LIN {X -0.165,Y -561.534,Z 1075.002,A 0.000,B 0.000,C 90.000,E1 36.457} C_DIS
LIN {X 0.132,Y -558.565,Z 1074.998,A 0.000,B 0.000,C 90.000,E1 35.598} C_DIS
LIN {X 0.308,Y -556.320,Z 1074.995,A 0.000,B 0.000,C 90.000,E1 35.025} C_DIS
LIN {X 0.102,Y -552.086,Z 1074.989,A 0.000,B 0.000,C 90.000,E1 34.072} C_DIS
LIN {X 0.098,Y -548.792,Z 1074.985,A 0.000,B 0.000,C 90.000,E1 33.372} C_DIS
LIN {X 0.057,Y -545.238,Z 1074.982,A 0.000,B 0.000,C 90.000,E1 32.673} C_DIS
LIN {X 0.305,Y -540.806,Z 1074.977,A 0.000,B 0.000,C 90.000,E1 31.799} C_DIS
LIN {X -0.096,Y -536.840,Z 1074.973,A 0.000,B 0.000,C 90.000,E1 31.131} C_DIS
LIN {X -0.067,Y -532.563,Z 1074.969,A 0.000,B 0.000,C 90.000,E1 30.413} C_DIS
LIN {X 0.077,Y -528.884,Z 1074.966,A 0.000,B 0.000,C 90.000,E1 29.823} C_DIS
LIN {X -0.264,Y -524.894,Z 1074.963,A 0.000,B 0.000,C 90.000,E1 29.283} C_DIS
LIN {X 0.207,Y -518.481,Z 1074.958,A 0.000,B 0.000,C 90.000,E1 28.359} C_DIS
LIN {X 0.070,Y -512.632,Z 1074.954,A 0.000,B 0.000,C 90.000,E1 27.641} C_DIS
LIN {X -0.093,Y -506.270,Z 1074.950,A 0.000,B 0.000,C 90.000,E1 26.924} C_DIS
LIN {X -0.260,Y -500.914,Z 1074.946,A 0.000,B 0.000,C 90.000,E1 26.360} C_DIS
LIN {X 0.212,Y -494.053,Z 1074.942,A 0.000,B 0.000,C 90.000,E1 25.591} C_DIS
LIN {X 0.027,Y -485.704,Z 1074.938,A 0.000,B 0.000,C 90.000,E1 24.771} C_DIS
LIN {X 0.015,Y -475.699,Z 1074.932,A 0.000,B 0.000,C 90.000,E1 23.823} C_DIS
LIN {X 0.046,Y -466.824,Z 1074.928,A 0.000,B 0.000,C 90.000,E1 23.025} C_DIS
LIN {X -0.178,Y -453.420,Z 1074.922,A 0.000,B 0.000,C 90.000,E1 21.897} C_DIS
LIN {X -0.124,Y -431.292,Z 1074.910,A 0.000,B 0.000,C 90.000,E1 19.885} C_DIS
LIN {X -0.144,Y -418.613,Z 1074.903,A 0.000,B 0.000,C 90.000,E1 18.598} C_DIS
LIN {X -0.076,Y -409.051,Z 1074.897,A 0.000,B 0.000,C 90.000,E1 17.511} C_DIS
LIN {X 0.161,Y -401.164,Z 1074.892,A 0.000,B 0.000,C 90.000,E1 16.496} C_DIS
LIN {X 0.146,Y -397.859,Z 1074.889,A 0.000,B 0.000,C 90.000,E1 16.024} C_DIS
LIN {X 0.115,Y -396.044,Z 1074.888,A 0.000,B 0.000,C 90.000,E1 15.733} C_DIS
LIN {X -0.218,Y -395.141,Z 1074.887,A 0.000,B 0.000,C 90.000,E1 15.607} C_DIS
LIN {X -0.143,Y -393.859,Z 1074.885,A 0.000,B 0.000,C 90.000,E1 15.245} C_DIS
LIN {X -0.113,Y -393.096,Z 1074.884,A 0.000,B 0.000,C 90.000,E1 15.064} C_DIS
LIN {X -0.139,Y -392.054,Z 1074.881,A 0.000,B 0.000,C 90.000,E1 14.537} C_DIS
LIN {X -0.159,Y -391.808,Z 1074.877,A 0.000,B 0.000,C 90.000,E1 13.828} C_DIS
LIN {X -0.069,Y -392.415,Z 1074.873,A 0.000,B 0.000,C 90.000,E1 13.119} C_DIS
LIN {X 0.034,Y -399.707,Z 1074.847,A 0.000,B 0.000,C 90.000,E1 8.511} C_DIS
LIN {X -0.090,Y -404.135,Z 1074.836,A 0.000,B 0.000,C 90.000,E1 6.429} C_DIS
LIN {X -0.169,Y -407.950,Z 1074.826,A 0.000,B 0.000,C 90.000,E1 4.702} C_DIS
LIN {X -0.197,Y -408.866,Z 1074.824,A 0.000,B 0.000,C 90.000,E1 4.359} C_DIS
LIN {X -0.189,Y -410.221,Z 1074.822,A 0.000,B 0.000,C 90.000,E1 4.012} C_DIS
LIN {X -0.001,Y -412.147,Z 1074.820,A 0.000,B 0.000,C 90.000,E1 3.555} C_DIS
LIN {X -0.190,Y -416.804,Z 1074.816,A 0.000,B 0.000,C 90.000,E1 2.980} C_DIS
LIN {X 0.020,Y -417.622,Z 1074.816,A 0.000,B 0.000,C 90.000,E1 2.865} C_DIS
LIN {X 0.179,Y -422.679,Z 1074.814,A 0.000,B 0.000,C 90.000,E1 2.465} C_DIS
LIN {X -0.036,Y -434.410,Z 1074.810,A 0.000,B 0.000,C 90.000,E1 1.718} C_DIS
LIN {X 0.080,Y -459.258,Z 1074.801,A 0.000,B 0.000,C 90.000,E1 0.115} C_DIS
LIN {X -0.087,Y -474.381,Z 1074.796,A 0.000,B 0.000,C 90.000,E1 359.198} C_DIS
LIN {X 0.111,Y -484.224,Z 1074.792,A 0.000,B 0.000,C 90.000,E1 358.568} C_DIS
LIN {X -0.207,Y -495.380,Z 1074.788,A 0.000,B 0.000,C 90.000,E1 357.879} C_DIS
LIN {X 0.115,Y -503.194,Z 1074.785,A 0.000,B 0.000,C 90.000,E1 357.306} C_DIS
LIN {X 0.058,Y -510.520,Z 1074.782,A 0.000,B 0.000,C 90.000,E1 356.788} C_DIS
LIN {X 0.050,Y -516.476,Z 1074.780,A 0.000,B 0.000,C 90.000,E1 356.331} C_DIS
LIN {X -0.225,Y -523.750,Z 1074.776,A 0.000,B 0.000,C 90.000,E1 355.755} C_DIS
LIN {X 0.086,Y -531.946,Z 1074.772,A 0.000,B 0.000,C 90.000,E1 354.951} C_DIS
LIN {X -0.076,Y -537.186,Z 1074.769,A 0.000,B 0.000,C 90.000,E1 354.432} C_DIS
LIN {X -0.184,Y -543.345,Z 1074.765,A 0.000,B 0.000,C 90.000,E1 353.742} C_DIS
LIN {X -0.095,Y -548.003,Z 1074.762,A 0.000,B 0.000,C 90.000,E1 353.166} C_DIS
LIN {X -0.159,Y -553.081,Z 1074.758,A 0.000,B 0.000,C 90.000,E1 352.470} C_DIS
LIN {X 0.000,Y -556.784,Z 1074.755,A 0.000,B 0.000,C 90.000,E1 351.894} C_DIS
LIN {X -0.228,Y -561.640,Z 1074.750,A 0.000,B 0.000,C 90.000,E1 351.084} C_DIS
LIN {X 0.232,Y -563.986,Z 1074.748,A 0.000,B 0.000,C 90.000,E1 350.622} C_DIS
LIN {X -0.071,Y -568.640,Z 1074.743,A 0.000,B 0.000,C 90.000,E1 349.690} C_DIS
LIN {X -0.268,Y -571.076,Z 1074.740,A 0.000,B 0.000,C 90.000,E1 349.162} C_DIS
LIN {X 0.308,Y -574.633,Z 1074.735,A 0.000,B 0.000,C 90.000,E1 348.285} C_DIS
LIN {X 0.232,Y -580.028,Z 1074.728,A 0.000,B 0.000,C 90.000,E1 346.937} C_DIS
LIN {X 0.003,Y -584.013,Z 1074.722,A 0.000,B 0.000,C 90.000,E1 345.880} C_DIS
LIN {X -0.029,Y -587.800,Z 1074.716,A 0.000,B 0.000,C 90.000,E1 344.810} C_DIS
LIN {X 0.307,Y -590.501,Z 1074.711,A 0.000,B 0.000,C 90.000,E1 343.976} C_DIS
LIN {X 0.059,Y -594.876,Z 1074.704,A 0.000,B 0.000,C 90.000,E1 342.670} C_DIS
LIN {X -0.217,Y -598.220,Z 1074.698,A 0.000,B 0.000,C 90.000,E1 341.638} C_DIS
LIN {X -0.347,Y -600.546,Z 1074.693,A 0.000,B 0.000,C 90.000,E1 340.859} C_DIS
LIN {X -0.064,Y -604.004,Z 1074.686,A 0.000,B 0.000,C 90.000,E1 339.518} C_DIS
LIN {X 0.067,Y -605.993,Z 1074.682,A 0.000,B 0.000,C 90.000,E1 338.720} C_DIS
LIN {X 0.216,Y -607.758,Z 1074.677,A 0.000,B 0.000,C 90.000,E1 337.922} C_DIS
LIN {X 0.286,Y -610.437,Z 1074.670,A 0.000,B 0.000,C 90.000,E1 336.613} C_DIS
LIN {X -0.161,Y -612.623,Z 1074.663,A 0.000,B 0.000,C 90.000,E1 335.357} C_DIS
LIN {X 0.243,Y -614.458,Z 1074.656,A 0.000,B 0.000,C 90.000,E1 334.024} C_DIS
LIN {X 0.149,Y -615.747,Z 1074.650,A 0.000,B 0.000,C 90.000,E1 332.999} C_DIS
LIN {X 0.087,Y -616.628,Z 1074.646,A 0.000,B 0.000,C 90.000,E1 332.231} C_DIS
LIN {X 0.290,Y -617.753,Z 1074.639,A 0.000,B 0.000,C 90.000,E1 330.923} C_DIS
LIN {X -0.008,Y -618.335,Z 1074.633,A 0.000,B 0.000,C 90.000,E1 329.921} C_DIS
LIN {X 0.237,Y -618.642,Z 1074.627,A 0.000,B 0.000,C 90.000,E1 328.869} C_DIS
LIN {X -0.028,Y -618.644,Z 1074.623,A 0.000,B 0.000,C 90.000,E1 328.122} C_DIS
LIN {X -0.011,Y -618.295,Z 1074.616,A 0.000,B 0.000,C 90.000,E1 326.834} C_DIS
LIN {X 0.030,Y -617.634,Z 1074.610,A 0.000,B 0.000,C 90.000,E1 325.801} C_DIS
LIN {X 0.102,Y -617.036,Z 1074.606,A 0.000,B 0.000,C 90.000,E1 325.022} C_DIS
LIN {X -0.013,Y -615.176,Z 1074.594,A 0.000,B 0.000,C 90.000,E1 322.970} C_DIS
LIN {X 0.069,Y -614.027,Z 1074.586,A 0.000,B 0.000,C 90.000,E1 321.412} C_DIS
LIN {X -0.062,Y -612.361,Z 1074.573,A 0.000,B 0.000,C 90.000,E1 319.094} C_DIS
LIN {X -0.035,Y -611.598,Z 1074.566,A 0.000,B 0.000,C 90.000,E1 317.796} C_DIS
LIN {X -0.388,Y -611.230,Z 1074.563,A 0.000,B 0.000,C 90.000,E1 317.310} C_DIS
LIN {X -0.323,Y -609.621,Z 1074.553,A 0.000,B 0.000,C 90.000,E1 315.486} C_DIS
LIN {X -0.060,Y -607.968,Z 1074.541,A 0.000,B 0.000,C 90.000,E1 313.380} C_DIS
LIN {X -0.301,Y -606.609,Z 1074.532,A 0.000,B 0.000,C 90.000,E1 311.838} C_DIS
LIN {X -0.108,Y -605.128,Z 1074.524,A 0.000,B 0.000,C 90.000,E1 310.253} C_DIS
LIN {X 0.001,Y -604.301,Z 1074.518,A 0.000,B 0.000,C 90.000,E1 309.197} C_DIS
LIN {X 0.049,Y -603.773,Z 1074.515,A 0.000,B 0.000,C 90.000,E1 308.669} C_DIS
LIN {X -0.025,Y -603.222,Z 1074.510,A 0.000,B 0.000,C 90.000,E1 307.890} C_DIS
LIN {X -0.408,Y -601.658,Z 1074.500,A 0.000,B 0.000,C 90.000,E1 306.091} C_DIS
LIN {X 0.341,Y -600.780,Z 1074.496,A 0.000,B 0.000,C 90.000,E1 305.231} C_DIS
LIN {X -0.102,Y -599.901,Z 1074.492,A 0.000,B 0.000,C 90.000,E1 304.485} C_DIS
LIN {X 0.158,Y -597.860,Z 1074.483,A 0.000,B 0.000,C 90.000,E1 302.880} C_DIS
LIN {X 0.197,Y -596.605,Z 1074.478,A 0.000,B 0.000,C 90.000,E1 302.084} C_DIS
LIN {X -0.183,Y -595.601,Z 1074.475,A 0.000,B 0.000,C 90.000,E1 301.592} C_DIS
LIN {X -0.163,Y -593.715,Z 1074.471,A 0.000,B 0.000,C 90.000,E1 300.797} C_DIS
LIN {X -0.160,Y -591.348,Z 1074.467,A 0.000,B 0.000,C 90.000,E1 300.001} C_DIS
LIN {X -0.182,Y -588.499,Z 1074.462,A 0.000,B 0.000,C 90.000,E1 299.205} C_DIS
LIN {X 0.217,Y -584.185,Z 1074.457,A 0.000,B 0.000,C 90.000,E1 298.231} C_DIS
LIN {X 0.032,Y -581.939,Z 1074.455,A 0.000,B 0.000,C 90.000,E1 297.847} C_DIS
LIN {X -0.163,Y -579.429,Z 1074.453,A 0.000,B 0.000,C 90.000,E1 297.462} C_DIS
LIN {X -0.178,Y -575.517,Z 1074.450,A 0.000,B 0.000,C 90.000,E1 296.924} C_DIS
LIN {X 0.185,Y -573.298,Z 1074.448,A 0.000,B 0.000,C 90.000,E1 296.616} C_DIS
LIN {X 0.109,Y -571.984,Z 1074.447,A 0.000,B 0.000,C 90.000,E1 296.488} C_DIS
LIN {X 0.021,Y -568.906,Z 1074.446,A 0.000,B 0.000,C 90.000,E1 296.232} C_DIS
LIN {X 0.165,Y -565.892,Z 1074.444,A 0.000,B 0.000,C 90.000,E1 295.976} C_DIS
LIN {X 0.274,Y -564.016,Z 1074.444,A 0.000,B 0.000,C 90.000,E1 295.848} C_DIS
LIN {X -0.123,Y -561.660,Z 1074.443,A 0.000,B 0.000,C 90.000,E1 295.771} C_DIS
LIN {X 0.029,Y -557.315,Z 1074.442,A 0.000,B 0.000,C 90.000,E1 295.591} C_DIS
LIN {X 0.071,Y -554.762,Z 1074.442,A 0.000,B 0.000,C 90.000,E1 295.463} C_DIS
LIN {X -0.158,Y -552.795,Z 1074.441,A 0.000,B 0.000,C 90.000,E1 295.412} C_DIS
LIN {X -0.148,Y -551.370,Z 1074.441,A 0.000,B 0.000,C 90.000,E1 295.335} C_DIS
LIN {X 0.171,Y -549.416,Z 1074.440,A 0.000,B 0.000,C 90.000,E1 295.155} C_DIS
LIN {X -0.319,Y -547.636,Z 1074.439,A 0.000,B 0.000,C 90.000,E1 295.027} C_DIS
LIN {X 0.122,Y -546.552,Z 1074.438,A 0.000,B 0.000,C 90.000,E1 294.847} C_DIS
LIN {X -0.055,Y -545.055,Z 1074.437,A 0.000,B 0.000,C 90.000,E1 294.591} C_DIS
LIN {X 0.068,Y -543.671,Z 1074.434,A 0.000,B 0.000,C 90.000,E1 294.155} C_DIS
LIN {X -0.264,Y -543.036,Z 1074.432,A 0.000,B 0.000,C 90.000,E1 293.770} C_DIS
LIN {X -0.282,Y -542.679,Z 1074.429,A 0.000,B 0.000,C 90.000,E1 293.206} C_DIS
LIN {X 0.170,Y -542.511,Z 1074.422,A 0.000,B 0.000,C 90.000,E1 292.025} C_DIS
LIN {X -0.088,Y -542.359,Z 1074.416,A 0.000,B 0.000,C 90.000,E1 290.918} C_DIS
LIN {X -0.060,Y -542.525,Z 1074.407,A 0.000,B 0.000,C 90.000,E1 289.214} C_DIS
LIN {X 0.186,Y -542.645,Z 1074.401,A 0.000,B 0.000,C 90.000,E1 288.055} C_DIS
LIN {X 0.259,Y -542.719,Z 1074.394,A 0.000,B 0.000,C 90.000,E1 286.913} C_DIS
LIN {X -0.121,Y -542.449,Z 1074.386,A 0.000,B 0.000,C 90.000,E1 285.536} C_DIS
LIN {X -0.128,Y -541.988,Z 1074.378,A 0.000,B 0.000,C 90.000,E1 284.120} C_DIS
LIN {X -0.143,Y -541.426,Z 1074.370,A 0.000,B 0.000,C 90.000,E1 282.703} C_DIS
LIN {X -0.215,Y -540.575,Z 1074.361,A 0.000,B 0.000,C 90.000,E1 281.007} C_DIS
LIN {X 0.198,Y -539.496,Z 1074.350,A 0.000,B 0.000,C 90.000,E1 278.973} C_DIS
LIN {X -0.094,Y -538.562,Z 1074.341,A 0.000,B 0.000,C 90.000,E1 277.296} C_DIS
LIN {X 0.069,Y -537.801,Z 1074.333,A 0.000,B 0.000,C 90.000,E1 275.853} C_DIS
LIN {X 0.207,Y -536.736,Z 1074.322,A 0.000,B 0.000,C 90.000,E1 273.841} C_DIS
LIN {X 0.259,Y -535.709,Z 1074.310,A 0.000,B 0.000,C 90.000,E1 271.835} C_DIS
LIN {X -0.247,Y -534.783,Z 1074.301,A 0.000,B 0.000,C 90.000,E1 270.172} C_DIS
LIN {X -0.249,Y -533.966,Z 1074.293,A 0.000,B 0.000,C 90.000,E1 268.740} C_DIS
LIN {X -0.248,Y -533.309,Z 1074.286,A 0.000,B 0.000,C 90.000,E1 267.593} C_DIS
LIN {X -0.242,Y -532.307,Z 1074.277,A 0.000,B 0.000,C 90.000,E1 265.869} C_DIS
LIN {X -0.240,Y -531.249,Z 1074.269,A 0.000,B 0.000,C 90.000,E1 264.432} C_DIS
LIN {X -0.205,Y -529.945,Z 1074.261,A 0.000,B 0.000,C 90.000,E1 262.989} C_DIS
LIN {X -0.196,Y -528.468,Z 1074.253,A 0.000,B 0.000,C 90.000,E1 261.546} C_DIS
LIN {X -0.093,Y -526.288,Z 1074.242,A 0.000,B 0.000,C 90.000,E1 259.511} C_DIS
LIN {X 0.050,Y -524.135,Z 1074.230,A 0.000,B 0.000,C 90.000,E1 257.465} C_DIS
LIN {X 0.230,Y -522.650,Z 1074.222,A 0.000,B 0.000,C 90.000,E1 255.992} C_DIS
LIN {X 0.008,Y -520.608,Z 1074.211,A 0.000,B 0.000,C 90.000,E1 253.976} C_DIS
LIN {X -0.111,Y -518.750,Z 1074.201,A 0.000,B 0.000,C 90.000,E1 252.236} C_DIS
LIN {X 0.111,Y -517.533,Z 1074.195,A 0.000,B 0.000,C 90.000,E1 251.040} C_DIS
LIN {X 0.122,Y -515.892,Z 1074.187,A 0.000,B 0.000,C 90.000,E1 249.571} C_DIS
LIN {X 0.104,Y -514.022,Z 1074.178,A 0.000,B 0.000,C 90.000,E1 248.103} C_DIS
LIN {X -0.116,Y -511.574,Z 1074.169,A 0.000,B 0.000,C 90.000,E1 246.357} C_DIS
LIN {X 0.181,Y -509.315,Z 1074.160,A 0.000,B 0.000,C 90.000,E1 244.845} C_DIS
LIN {X -0.026,Y -506.957,Z 1074.152,A 0.000,B 0.000,C 90.000,E1 243.384} C_DIS
LIN {X 0.320,Y -504.954,Z 1074.146,A 0.000,B 0.000,C 90.000,E1 242.153} C_DIS
LIN {X 0.121,Y -501.896,Z 1074.136,A 0.000,B 0.000,C 90.000,E1 240.383} C_DIS
LIN {X -0.154,Y -498.729,Z 1074.126,A 0.000,B 0.000,C 90.000,E1 238.614} C_DIS
LIN {X 0.006,Y -495.417,Z 1074.115,A 0.000,B 0.000,C 90.000,E1 236.786} C_DIS
LIN {X -0.048,Y -491.856,Z 1074.105,A 0.000,B 0.000,C 90.000,E1 234.975} C_DIS
LIN {X 0.265,Y -488.776,Z 1074.097,A 0.000,B 0.000,C 90.000,E1 233.417} C_DIS
LIN {X 0.127,Y -485.562,Z 1074.089,A 0.000,B 0.000,C 90.000,E1 231.904} C_DIS
LIN {X 0.043,Y -481.501,Z 1074.078,A 0.000,B 0.000,C 90.000,E1 230.070} C_DIS
LIN {X -0.183,Y -475.565,Z 1074.063,A 0.000,B 0.000,C 90.000,E1 227.310} C_DIS
LIN {X -0.052,Y -470.828,Z 1074.049,A 0.000,B 0.000,C 90.000,E1 224.798} C_DIS
LIN {X 0.034,Y -467.996,Z 1074.040,A 0.000,B 0.000,C 90.000,E1 223.218} C_DIS
LIN {X -0.248,Y -464.960,Z 1074.031,A 0.000,B 0.000,C 90.000,E1 221.676} C_DIS
LIN {X 0.161,Y -461.136,Z 1074.021,A 0.000,B 0.000,C 90.000,E1 219.725} C_DIS
LIN {X -0.192,Y -458.057,Z 1074.012,A 0.000,B 0.000,C 90.000,E1 218.177} C_DIS
LIN {X -0.244,Y -454.887,Z 1074.003,A 0.000,B 0.000,C 90.000,E1 216.583} C_DIS
LIN {X -0.204,Y -450.241,Z 1073.991,A 0.000,B 0.000,C 90.000,E1 214.326} C_DIS
LIN {X 0.198,Y -445.779,Z 1073.978,A 0.000,B 0.000,C 90.000,E1 212.005} C_DIS
LIN {X 0.071,Y -443.385,Z 1073.971,A 0.000,B 0.000,C 90.000,E1 210.718} C_DIS
LIN {X 0.111,Y -440.255,Z 1073.962,A 0.000,B 0.000,C 90.000,E1 209.077} C_DIS
LIN {X -0.087,Y -436.535,Z 1073.951,A 0.000,B 0.000,C 90.000,E1 207.129} C_DIS
LIN {X -0.175,Y -433.150,Z 1073.940,A 0.000,B 0.000,C 90.000,E1 205.155} C_DIS
LIN {X -0.144,Y -429.512,Z 1073.927,A 0.000,B 0.000,C 90.000,E1 202.823} C_DIS
LIN {X 0.044,Y -426.761,Z 1073.916,A 0.000,B 0.000,C 90.000,E1 200.791} C_DIS
LIN {X -0.162,Y -425.837,Z 1073.910,A 0.000,B 0.000,C 90.000,E1 199.812} C_DIS
LIN {X -0.173,Y -425.484,Z 1073.906,A 0.000,B 0.000,C 90.000,E1 199.141} C_DIS
LIN {X 0.215,Y -425.212,Z 1073.902,A 0.000,B 0.000,C 90.000,E1 198.417} C_DIS
LIN {X 0.065,Y -425.334,Z 1073.899,A 0.000,B 0.000,C 90.000,E1 197.764} C_DIS
LIN {X 0.046,Y -425.808,Z 1073.895,A 0.000,B 0.000,C 90.000,E1 197.094} C_DIS
LIN {X -0.097,Y -426.809,Z 1073.891,A 0.000,B 0.000,C 90.000,E1 196.441} C_DIS
LIN {X -0.031,Y -429.236,Z 1073.886,A 0.000,B 0.000,C 90.000,E1 195.426} C_DIS
LIN {X -0.044,Y -431.990,Z 1073.881,A 0.000,B 0.000,C 90.000,E1 194.592} C_DIS
LIN {X 0.006,Y -439.992,Z 1073.871,A 0.000,B 0.000,C 90.000,E1 192.771} C_DIS
LIN {X -0.216,Y -450.151,Z 1073.860,A 0.000,B 0.000,C 90.000,E1 190.838} C_DIS
LIN {X 0.164,Y -461.062,Z 1073.849,A 0.000,B 0.000,C 90.000,E1 188.859} C_DIS
LIN {X 0.192,Y -468.397,Z 1073.842,A 0.000,B 0.000,C 90.000,E1 187.587} C_DIS
LIN {X 0.039,Y -473.849,Z 1073.837,A 0.000,B 0.000,C 90.000,E1 186.663} C_DIS
LIN {X -0.057,Y -479.015,Z 1073.832,A 0.000,B 0.000,C 90.000,E1 185.739} C_DIS
LIN {X 0.044,Y -484.844,Z 1073.826,A 0.000,B 0.000,C 90.000,E1 184.645} C_DIS
LIN {X 0.026,Y -489.888,Z 1073.821,A 0.000,B 0.000,C 90.000,E1 183.726} C_DIS
LIN {X 0.238,Y -495.579,Z 1073.815,A 0.000,B 0.000,C 90.000,E1 182.636} C_DIS
LIN {X 0.028,Y -501.228,Z 1073.809,A 0.000,B 0.000,C 90.000,E1 181.604} C_DIS
LIN {X 0.075,Y -507.486,Z 1073.802,A 0.000,B 0.000,C 90.000,E1 180.401} C_DIS
LIN {X 0.142,Y -515.276,Z 1073.794,A 0.000,B 0.000,C 90.000,E1 178.912} C_DIS
LIN {X 0.184,Y -520.701,Z 1073.788,A 0.000,B 0.000,C 90.000,E1 177.879} C_DIS
LIN {X -0.044,Y -529.758,Z 1073.779,A 0.000,B 0.000,C 90.000,E1 176.159} C_DIS
LIN {X -0.007,Y -538.730,Z 1073.769,A 0.000,B 0.000,C 90.000,E1 174.432} C_DIS
LIN {X -0.051,Y -546.842,Z 1073.760,A 0.000,B 0.000,C 90.000,E1 172.875} C_DIS
LIN {X 0.198,Y -552.617,Z 1073.754,A 0.000,B 0.000,C 90.000,E1 171.724} C_DIS
LIN {X 0.055,Y -558.314,Z 1073.748,A 0.000,B 0.000,C 90.000,E1 170.622} C_DIS
LIN {X -0.160,Y -564.503,Z 1073.741,A 0.000,B 0.000,C 90.000,E1 169.398} C_DIS
LIN {X 0.102,Y -569.230,Z 1073.736,A 0.000,B 0.000,C 90.000,E1 168.409} C_DIS
LIN {X 0.100,Y -573.086,Z 1073.731,A 0.000,B 0.000,C 90.000,E1 167.589} C_DIS
LIN {X -0.211,Y -580.574,Z 1073.722,A 0.000,B 0.000,C 90.000,E1 165.992} C_DIS
LIN {X -0.191,Y -584.733,Z 1073.717,A 0.000,B 0.000,C 90.000,E1 165.046} C_DIS
LIN {X 0.111,Y -588.117,Z 1073.712,A 0.000,B 0.000,C 90.000,E1 164.212} C_DIS
LIN {X 0.141,Y -592.450,Z 1073.706,A 0.000,B 0.000,C 90.000,E1 163.142} C_DIS
LIN {X -0.042,Y -595.527,Z 1073.702,A 0.000,B 0.000,C 90.000,E1 162.362} C_DIS
LIN {X 0.264,Y -599.459,Z 1073.696,A 0.000,B 0.000,C 90.000,E1 161.275} C_DIS
LIN {X -0.232,Y -604.018,Z 1073.689,A 0.000,B 0.000,C 90.000,E1 160.007} C_DIS
LIN {X -0.103,Y -606.577,Z 1073.684,A 0.000,B 0.000,C 90.000,E1 159.209} C_DIS
LIN {X -0.280,Y -610.636,Z 1073.677,A 0.000,B 0.000,C 90.000,E1 157.922} C_DIS
LIN {X 0.151,Y -613.007,Z 1073.673,A 0.000,B 0.000,C 90.000,E1 157.102} C_DIS
LIN {X 0.319,Y -616.607,Z 1073.666,A 0.000,B 0.000,C 90.000,E1 155.793} C_DIS
LIN {X -0.030,Y -620.754,Z 1073.657,A 0.000,B 0.000,C 90.000,E1 154.280} C_DIS
LIN {X -0.031,Y -624.543,Z 1073.649,A 0.000,B 0.000,C 90.000,E1 152.743} C_DIS
LIN {X 0.007,Y -627.078,Z 1073.643,A 0.000,B 0.000,C 90.000,E1 151.719} C_DIS
LIN {X -0.174,Y -629.490,Z 1073.637,A 0.000,B 0.000,C 90.000,E1 150.717} C_DIS
LIN {X -0.259,Y -632.942,Z 1073.629,A 0.000,B 0.000,C 90.000,E1 149.203} C_DIS
LIN {X 0.074,Y -636.745,Z 1073.619,A 0.000,B 0.000,C 90.000,E1 147.406} C_DIS
LIN {X -0.238,Y -640.357,Z 1073.609,A 0.000,B 0.000,C 90.000,E1 145.674} C_DIS
LIN {X 0.018,Y -643.392,Z 1073.601,A 0.000,B 0.000,C 90.000,E1 144.149} C_DIS
LIN {X 0.189,Y -646.342,Z 1073.593,A 0.000,B 0.000,C 90.000,E1 142.637} C_DIS
LIN {X 0.045,Y -647.872,Z 1073.588,A 0.000,B 0.000,C 90.000,E1 141.904} C_DIS
LIN {X 0.281,Y -650.336,Z 1073.582,A 0.000,B 0.000,C 90.000,E1 140.642} C_DIS
LIN {X 0.030,Y -653.843,Z 1073.572,A 0.000,B 0.000,C 90.000,E1 138.933} C_DIS
LIN {X -0.173,Y -656.959,Z 1073.564,A 0.000,B 0.000,C 90.000,E1 137.472} C_DIS
LIN {X 0.089,Y -661.271,Z 1073.553,A 0.000,B 0.000,C 90.000,E1 135.486} C_DIS
LIN {X 0.009,Y -664.876,Z 1073.545,A 0.000,B 0.000,C 90.000,E1 134.028} C_DIS
LIN {X 0.028,Y -669.235,Z 1073.535,A 0.000,B 0.000,C 90.000,E1 132.324} C_DIS
LIN {X 0.138,Y -673.000,Z 1073.527,A 0.000,B 0.000,C 90.000,E1 130.862} C_DIS
LIN {X -0.123,Y -676.778,Z 1073.519,A 0.000,B 0.000,C 90.000,E1 129.439} C_DIS
LIN {X -0.158,Y -681.668,Z 1073.508,A 0.000,B 0.000,C 90.000,E1 127.523} C_DIS
LIN {X -0.342,Y -684.154,Z 1073.503,A 0.000,B 0.000,C 90.000,E1 126.583} C_DIS
LIN {X -0.124,Y -686.021,Z 1073.499,A 0.000,B 0.000,C 90.000,E1 125.851} C_DIS
LIN {X -0.079,Y -688.857,Z 1073.493,A 0.000,B 0.000,C 90.000,E1 124.659} C_DIS
LIN {X 0.203,Y -691.761,Z 1073.486,A 0.000,B 0.000,C 90.000,E1 123.452} C_DIS
LIN {X -0.266,Y -694.068,Z 1073.481,A 0.000,B 0.000,C 90.000,E1 122.546} C_DIS
LIN {X 0.223,Y -695.750,Z 1073.477,A 0.000,B 0.000,C 90.000,E1 121.799} C_DIS
LIN {X -0.324,Y -698.389,Z 1073.470,A 0.000,B 0.000,C 90.000,E1 120.669} C_DIS
LIN {X 0.201,Y -699.820,Z 1073.466,A 0.000,B 0.000,C 90.000,E1 119.922} C_DIS
LIN {X 0.391,Y -700.876,Z 1073.463,A 0.000,B 0.000,C 90.000,E1 119.205} C_DIS
LIN {X 0.318,Y -701.494,Z 1073.460,A 0.000,B 0.000,C 90.000,E1 118.743} C_DIS
LIN {X 0.002,Y -703.478,Z 1073.448,A 0.000,B 0.000,C 90.000,E1 116.668} C_DIS
LIN {X 0.194,Y -704.395,Z 1073.443,A 0.000,B 0.000,C 90.000,E1 115.720} C_DIS
LIN {X -0.173,Y -704.786,Z 1073.440,A 0.000,B 0.000,C 90.000,E1 115.283} C_DIS
LIN {X -0.238,Y -704.963,Z 1073.438,A 0.000,B 0.000,C 90.000,E1 114.823} C_DIS
LIN {X -0.245,Y -704.961,Z 1073.437,A 0.000,B 0.000,C 90.000,E1 114.591} C_DIS
LIN {X 0.328,Y -704.505,Z 1073.434,A 0.000,B 0.000,C 90.000,E1 114.079} C_DIS
LIN {X -0.316,Y -703.985,Z 1073.433,A 0.000,B 0.000,C 90.000,E1 113.898} C_DIS
LIN {X 0.248,Y -702.448,Z 1073.430,A 0.000,B 0.000,C 90.000,E1 113.387} C_DIS
LIN {X 0.386,Y -701.844,Z 1073.429,A 0.000,B 0.000,C 90.000,E1 113.259} C_DIS
LIN {X 0.007,Y -698.300,Z 1073.427,A 0.000,B 0.000,C 90.000,E1 112.823} C_DIS
LIN {X -0.131,Y -697.259,Z 1073.426,A 0.000,B 0.000,C 90.000,E1 112.717} C_DIS
LIN {X -0.001,Y -695.687,Z 1073.426,A 0.000,B 0.000,C 90.000,E1 112.589} C_DIS
LIN {X -0.164,Y -688.279,Z 1073.424,A 0.000,B 0.000,C 90.000,E1 112.259} C_DIS
LIN {X 0.227,Y -686.446,Z 1073.423,A 0.000,B 0.000,C 90.000,E1 112.153} C_DIS
LIN {X 0.128,Y -684.148,Z 1073.423,A 0.000,B 0.000,C 90.000,E1 112.099} C_DIS
LIN {X -0.175,Y -676.156,Z 1073.422,A 0.000,B 0.000,C 90.000,E1 112.025} C_DIS
LIN {X -0.205,Y -607.048,Z 1073.422,A 0.000,B 0.000,C 90.000,E1 112.025} C_DIS
LIN {X 0.255,Y -601.997,Z 1073.421,A 0.000,B 0.000,C 90.000,E1 111.770} C_DIS
LIN {X 0.315,Y -596.175,Z 1073.419,A 0.000,B 0.000,C 90.000,E1 111.408} C_DIS
LIN {X 0.074,Y -588.927,Z 1073.416,A 0.000,B 0.000,C 90.000,E1 110.865} C_DIS
LIN {X 0.166,Y -580.721,Z 1073.412,A 0.000,B 0.000,C 90.000,E1 110.174} C_DIS
LIN {X 0.161,Y -575.155,Z 1073.410,A 0.000,B 0.000,C 90.000,E1 109.704} C_DIS
LIN {X 0.085,Y -569.130,Z 1073.407,A 0.000,B 0.000,C 90.000,E1 109.268} C_DIS
LIN {X -0.122,Y -560.870,Z 1073.404,A 0.000,B 0.000,C 90.000,E1 108.779} C_DIS
LIN {X -0.172,Y -554.271,Z 1073.402,A 0.000,B 0.000,C 90.000,E1 108.417} C_DIS
LIN {X 0.050,Y -549.376,Z 1073.400,A 0.000,B 0.000,C 90.000,E1 108.055} C_DIS
LIN {X -0.163,Y -547.701,Z 1073.399,A 0.000,B 0.000,C 90.000,E1 107.873} C_DIS
LIN {X -0.205,Y -547.669,Z 1073.399,A 0.000,B 0.000,C 90.000,E1 107.873} C_DIS
LIN {X -0.176,Y -547.352,Z 1073.398,A 0.000,B 0.000,C 90.000,E1 107.638} C_DIS
LIN {X 0.157,Y -547.444,Z 1073.395,A 0.000,B 0.000,C 90.000,E1 107.040} C_DIS
LIN {X -0.130,Y -548.416,Z 1073.387,A 0.000,B 0.000,C 90.000,E1 105.662} C_DIS
LIN {X -0.105,Y -549.993,Z 1073.375,A 0.000,B 0.000,C 90.000,E1 103.411} C_DIS
LIN {X 0.256,Y -551.925,Z 1073.362,A 0.000,B 0.000,C 90.000,E1 101.130} C_DIS
LIN {X 0.034,Y -554.290,Z 1073.350,A 0.000,B 0.000,C 90.000,E1 98.916} C_DIS
LIN {X 0.073,Y -556.176,Z 1073.340,A 0.000,B 0.000,C 90.000,E1 97.239} C_DIS
LIN {X 0.020,Y -557.718,Z 1073.333,A 0.000,B 0.000,C 90.000,E1 95.853} C_DIS
LIN {X -0.066,Y -559.077,Z 1073.325,A 0.000,B 0.000,C 90.000,E1 94.473} C_DIS
LIN {X -0.132,Y -559.941,Z 1073.317,A 0.000,B 0.000,C 90.000,E1 93.094} C_DIS
LIN {X -0.220,Y -560.677,Z 1073.309,A 0.000,B 0.000,C 90.000,E1 91.718} C_DIS
LIN {X -0.208,Y -561.466,Z 1073.300,A 0.000,B 0.000,C 90.000,E1 90.057} C_DIS
LIN {X -0.180,Y -562.039,Z 1073.291,A 0.000,B 0.000,C 90.000,E1 88.396} C_DIS
LIN {X -0.101,Y -562.696,Z 1073.282,A 0.000,B 0.000,C 90.000,E1 86.731} C_DIS
LIN {X -0.139,Y -563.235,Z 1073.274,A 0.000,B 0.000,C 90.000,E1 85.355} C_DIS
LIN {X 0.015,Y -563.758,Z 1073.265,A 0.000,B 0.000,C 90.000,E1 83.685} C_DIS
LIN {X 0.252,Y -564.259,Z 1073.256,A 0.000,B 0.000,C 90.000,E1 82.008} C_DIS
LIN {X 0.171,Y -564.524,Z 1073.250,A 0.000,B 0.000,C 90.000,E1 80.914} C_DIS
LIN {X -0.116,Y -565.090,Z 1073.242,A 0.000,B 0.000,C 90.000,E1 79.567} C_DIS
LIN {X 0.233,Y -565.824,Z 1073.233,A 0.000,B 0.000,C 90.000,E1 77.881} C_DIS
LIN {X -0.098,Y -566.875,Z 1073.222,A 0.000,B 0.000,C 90.000,E1 75.992} C_DIS
LIN {X 0.044,Y -568.982,Z 1073.205,A 0.000,B 0.000,C 90.000,E1 72.960} C_DIS
LIN {X 0.099,Y -570.513,Z 1073.195,A 0.000,B 0.000,C 90.000,E1 71.040} C_DIS
LIN {X 0.032,Y -572.135,Z 1073.184,A 0.000,B 0.000,C 90.000,E1 69.135} C_DIS
LIN {X 0.010,Y -573.674,Z 1073.174,A 0.000,B 0.000,C 90.000,E1 67.230} C_DIS
LIN {X -0.136,Y -574.960,Z 1073.165,A 0.000,B 0.000,C 90.000,E1 65.613} C_DIS
LIN {X -0.026,Y -575.984,Z 1073.155,A 0.000,B 0.000,C 90.000,E1 63.973} C_DIS
LIN {X -0.159,Y -576.937,Z 1073.146,A 0.000,B 0.000,C 90.000,E1 62.359} C_DIS
LIN {X 0.006,Y -577.832,Z 1073.137,A 0.000,B 0.000,C 90.000,E1 60.717} C_DIS
LIN {X 0.341,Y -578.490,Z 1073.130,A 0.000,B 0.000,C 90.000,E1 59.331} C_DIS
LIN {X 0.186,Y -579.098,Z 1073.122,A 0.000,B 0.000,C 90.000,E1 57.995} C_DIS
LIN {X 0.190,Y -579.849,Z 1073.113,A 0.000,B 0.000,C 90.000,E1 56.373} C_DIS
LIN {X 0.044,Y -580.513,Z 1073.104,A 0.000,B 0.000,C 90.000,E1 54.769} C_DIS
LIN {X -0.090,Y -580.799,Z 1073.098,A 0.000,B 0.000,C 90.000,E1 53.703} C_DIS
LIN {X -0.050,Y -581.040,Z 1073.091,A 0.000,B 0.000,C 90.000,E1 52.351} C_DIS
LIN {X 0.006,Y -580.977,Z 1073.086,A 0.000,B 0.000,C 90.000,E1 51.537} C_DIS
LIN {X 0.064,Y -580.869,Z 1073.082,A 0.000,B 0.000,C 90.000,E1 50.723} C_DIS
LIN {X 0.009,Y -580.452,Z 1073.074,A 0.000,B 0.000,C 90.000,E1 49.380} C_DIS
LIN {X -0.219,Y -580.027,Z 1073.068,A 0.000,B 0.000,C 90.000,E1 48.324} C_DIS
LIN {X -0.067,Y -579.457,Z 1073.062,A 0.000,B 0.000,C 90.000,E1 47.229} C_DIS
LIN {X -0.198,Y -578.610,Z 1073.055,A 0.000,B 0.000,C 90.000,E1 45.891} C_DIS
LIN {X -0.074,Y -577.673,Z 1073.049,A 0.000,B 0.000,C 90.000,E1 44.798} C_DIS
LIN {X 0.318,Y -576.792,Z 1073.044,A 0.000,B 0.000,C 90.000,E1 43.947} C_DIS
LIN {X 0.000,Y -575.375,Z 1073.038,A 0.000,B 0.000,C 90.000,E1 42.894} C_DIS
LIN {X 0.211,Y -573.401,Z 1073.031,A 0.000,B 0.000,C 90.000,E1 41.515} C_DIS
LIN {X -0.117,Y -571.371,Z 1073.025,A 0.000,B 0.000,C 90.000,E1 40.458} C_DIS
LIN {X 0.147,Y -570.322,Z 1073.022,A 0.000,B 0.000,C 90.000,E1 39.886} C_DIS
LIN {X -0.221,Y -567.791,Z 1073.016,A 0.000,B 0.000,C 90.000,E1 38.830} C_DIS
LIN {X 0.144,Y -565.719,Z 1073.011,A 0.000,B 0.000,C 90.000,E1 37.971} C_DIS
LIN {X 0.039,Y -563.336,Z 1073.006,A 0.000,B 0.000,C 90.000,E1 37.156} C_DIS
LIN {X 0.252,Y -561.570,Z 1073.003,A 0.000,B 0.000,C 90.000,E1 36.583} C_DIS
LIN {X -0.144,Y -557.497,Z 1072.997,A 0.000,B 0.000,C 90.000,E1 35.518} C_DIS
LIN {X -0.022,Y -553.378,Z 1072.992,A 0.000,B 0.000,C 90.000,E1 34.532} C_DIS
LIN {X -0.017,Y -550.202,Z 1072.988,A 0.000,B 0.000,C 90.000,E1 33.833} C_DIS
LIN {X -0.217,Y -547.505,Z 1072.985,A 0.000,B 0.000,C 90.000,E1 33.293} C_DIS
LIN {X 0.059,Y -543.151,Z 1072.980,A 0.000,B 0.000,C 90.000,E1 32.418} C_DIS
LIN {X -0.036,Y -539.405,Z 1072.976,A 0.000,B 0.000,C 90.000,E1 31.720} C_DIS
LIN {X 0.012,Y -535.355,Z 1072.972,A 0.000,B 0.000,C 90.000,E1 31.003} C_DIS
LIN {X -0.285,Y -531.891,Z 1072.969,A 0.000,B 0.000,C 90.000,E1 30.463} C_DIS
LIN {X -0.147,Y -528.175,Z 1072.966,A 0.000,B 0.000,C 90.000,E1 29.873} C_DIS
LIN {X -0.037,Y -524.183,Z 1072.963,A 0.000,B 0.000,C 90.000,E1 29.283} C_DIS
LIN {X -0.033,Y -517.759,Z 1072.958,A 0.000,B 0.000,C 90.000,E1 28.409} C_DIS
LIN {X 0.276,Y -511.837,Z 1072.954,A 0.000,B 0.000,C 90.000,E1 27.641} C_DIS
LIN {X -0.091,Y -504.144,Z 1072.949,A 0.000,B 0.000,C 90.000,E1 26.796} C_DIS
LIN {X -0.007,Y -495.954,Z 1072.944,A 0.000,B 0.000,C 90.000,E1 25.924} C_DIS
LIN {X 0.084,Y -487.798,Z 1072.939,A 0.000,B 0.000,C 90.000,E1 25.079} C_DIS
LIN {X -0.004,Y -477.835,Z 1072.934,A 0.000,B 0.000,C 90.000,E1 24.131} C_DIS
LIN {X -0.123,Y -468.857,Z 1072.930,A 0.000,B 0.000,C 90.000,E1 23.334} C_DIS
LIN {X 0.162,Y -461.299,Z 1072.926,A 0.000,B 0.000,C 90.000,E1 22.642} C_DIS
LIN {X 0.095,Y -446.431,Z 1072.919,A 0.000,B 0.000,C 90.000,E1 21.354} C_DIS
LIN {X 0.075,Y -431.541,Z 1072.911,A 0.000,B 0.000,C 90.000,E1 19.993} C_DIS
LIN {X 0.101,Y -418.552,Z 1072.904,A 0.000,B 0.000,C 90.000,E1 18.671} C_DIS
LIN {X 0.005,Y -410.301,Z 1072.899,A 0.000,B 0.000,C 90.000,E1 17.764} C_DIS
LIN {X 0.128,Y -402.103,Z 1072.893,A 0.000,B 0.000,C 90.000,E1 16.749} C_DIS
LIN {X 0.197,Y -397.437,Z 1072.890,A 0.000,B 0.000,C 90.000,E1 16.079} C_DIS
LIN {X 0.086,Y -394.908,Z 1072.887,A 0.000,B 0.000,C 90.000,E1 15.662} C_DIS
LIN {X -0.039,Y -392.898,Z 1072.884,A 0.000,B 0.000,C 90.000,E1 15.134} C_DIS
LIN {X -0.107,Y -391.937,Z 1072.881,A 0.000,B 0.000,C 90.000,E1 14.592} C_DIS
LIN {X -0.118,Y -391.858,Z 1072.877,A 0.000,B 0.000,C 90.000,E1 13.883} C_DIS
LIN {X -0.200,Y -392.705,Z 1072.872,A 0.000,B 0.000,C 90.000,E1 13.008} C_DIS
LIN {X -0.071,Y -400.055,Z 1072.847,A 0.000,B 0.000,C 90.000,E1 8.398} C_DIS
LIN {X 0.216,Y -405.226,Z 1072.833,A 0.000,B 0.000,C 90.000,E1 5.910} C_DIS
LIN {X 0.152,Y -408.297,Z 1072.825,A 0.000,B 0.000,C 90.000,E1 4.531} C_DIS
LIN {X 0.128,Y -409.217,Z 1072.823,A 0.000,B 0.000,C 90.000,E1 4.188} C_DIS
LIN {X 0.126,Y -412.208,Z 1072.820,A 0.000,B 0.000,C 90.000,E1 3.498} C_DIS
LIN {X 0.165,Y -416.970,Z 1072.816,A 0.000,B 0.000,C 90.000,E1 2.865} C_DIS
LIN {X 0.168,Y -418.957,Z 1072.815,A 0.000,B 0.000,C 90.000,E1 2.694} C_DIS
LIN {X 0.035,Y -422.208,Z 1072.814,A 0.000,B 0.000,C 90.000,E1 2.465} C_DIS
LIN {X 0.163,Y -436.652,Z 1072.808,A 0.000,B 0.000,C 90.000,E1 1.489} C_DIS
LIN {X 0.000,Y -460.447,Z 1072.800,A 0.000,B 0.000,C 90.000,E1 360.000} C_DIS
LIN {X -0.073,Y -473.589,Z 1072.796,A 0.000,B 0.000,C 90.000,E1 359.198} C_DIS
LIN {X 0.119,Y -483.494,Z 1072.792,A 0.000,B 0.000,C 90.000,E1 358.568} C_DIS
LIN {X -0.216,Y -492.957,Z 1072.789,A 0.000,B 0.000,C 90.000,E1 357.993} C_DIS
LIN {X 0.121,Y -499.203,Z 1072.786,A 0.000,B 0.000,C 90.000,E1 357.535} C_DIS
LIN {X -0.073,Y -508.597,Z 1072.783,A 0.000,B 0.000,C 90.000,E1 356.906} C_DIS
LIN {X -0.028,Y -517.485,Z 1072.779,A 0.000,B 0.000,C 90.000,E1 356.216} C_DIS
LIN {X -0.240,Y -523.380,Z 1072.776,A 0.000,B 0.000,C 90.000,E1 355.755} C_DIS
LIN {X 0.129,Y -531.582,Z 1072.772,A 0.000,B 0.000,C 90.000,E1 354.951} C_DIS
LIN {X -0.189,Y -538.061,Z 1072.768,A 0.000,B 0.000,C 90.000,E1 354.318} C_DIS
LIN {X 0.252,Y -544.199,Z 1072.765,A 0.000,B 0.000,C 90.000,E1 353.571} C_DIS
LIN {X 0.067,Y -547.723,Z 1072.762,A 0.000,B 0.000,C 90.000,E1 353.166} C_DIS
LIN {X 0.002,Y -552.872,Z 1072.758,A 0.000,B 0.000,C 90.000,E1 352.470} C_DIS
LIN {X -0.090,Y -557.474,Z 1072.754,A 0.000,B 0.000,C 90.000,E1 351.781} C_DIS
LIN {X -0.067,Y -561.536,Z 1072.750,A 0.000,B 0.000,C 90.000,E1 351.084} C_DIS
LIN {X 0.240,Y -564.599,Z 1072.747,A 0.000,B 0.000,C 90.000,E1 350.500} C_DIS
LIN {X -0.048,Y -569.279,Z 1072.742,A 0.000,B 0.000,C 90.000,E1 349.567} C_DIS
LIN {X -0.089,Y -574.681,Z 1072.735,A 0.000,B 0.000,C 90.000,E1 348.342} C_DIS
LIN {X 0.182,Y -579.069,Z 1072.729,A 0.000,B 0.000,C 90.000,E1 347.229} C_DIS
LIN {X -0.057,Y -583.196,Z 1072.723,A 0.000,B 0.000,C 90.000,E1 346.172} C_DIS
LIN {X -0.099,Y -587.040,Z 1072.717,A 0.000,B 0.000,C 90.000,E1 345.102} C_DIS
LIN {X -0.084,Y -590.699,Z 1072.711,A 0.000,B 0.000,C 90.000,E1 344.031} C_DIS
LIN {X -0.327,Y -595.132,Z 1072.704,A 0.000,B 0.000,C 90.000,E1 342.725} C_DIS
LIN {X -0.030,Y -598.463,Z 1072.698,A 0.000,B 0.000,C 90.000,E1 341.638} C_DIS
LIN {X -0.158,Y -600.826,Z 1072.694,A 0.000,B 0.000,C 90.000,E1 340.859} C_DIS
LIN {X 0.132,Y -604.344,Z 1072.686,A 0.000,B 0.000,C 90.000,E1 339.518} C_DIS
LIN {X 0.266,Y -606.327,Z 1072.682,A 0.000,B 0.000,C 90.000,E1 338.720} C_DIS
LIN {X -0.143,Y -608.151,Z 1072.678,A 0.000,B 0.000,C 90.000,E1 337.975} C_DIS
LIN {X 0.029,Y -609.782,Z 1072.673,A 0.000,B 0.000,C 90.000,E1 337.177} C_DIS
LIN {X -0.106,Y -611.329,Z 1072.669,A 0.000,B 0.000,C 90.000,E1 336.410} C_DIS
LIN {X 0.059,Y -613.081,Z 1072.663,A 0.000,B 0.000,C 90.000,E1 335.357} C_DIS
LIN {X -0.081,Y -614.946,Z 1072.656,A 0.000,B 0.000,C 90.000,E1 334.076} C_DIS
LIN {X -0.165,Y -616.285,Z 1072.650,A 0.000,B 0.000,C 90.000,E1 333.050} C_DIS
LIN {X -0.235,Y -617.437,Z 1072.645,A 0.000,B 0.000,C 90.000,E1 332.025} C_DIS
LIN {X -0.013,Y -618.532,Z 1072.637,A 0.000,B 0.000,C 90.000,E1 330.717} C_DIS
LIN {X -0.058,Y -619.004,Z 1072.633,A 0.000,B 0.000,C 90.000,E1 329.950} C_DIS
LIN {X -0.024,Y -619.382,Z 1072.627,A 0.000,B 0.000,C 90.000,E1 328.918} C_DIS
LIN {X 0.228,Y -619.436,Z 1072.622,A 0.000,B 0.000,C 90.000,E1 327.867} C_DIS
LIN {X -0.264,Y -619.079,Z 1072.615,A 0.000,B 0.000,C 90.000,E1 326.628} C_DIS
LIN {X -0.213,Y -618.494,Z 1072.609,A 0.000,B 0.000,C 90.000,E1 325.595} C_DIS
LIN {X -0.131,Y -617.951,Z 1072.604,A 0.000,B 0.000,C 90.000,E1 324.815} C_DIS
LIN {X -0.223,Y -616.269,Z 1072.593,A 0.000,B 0.000,C 90.000,E1 322.763} C_DIS
LIN {X -0.043,Y -615.408,Z 1072.586,A 0.000,B 0.000,C 90.000,E1 321.457} C_DIS
LIN {X -0.181,Y -614.596,Z 1072.580,A 0.000,B 0.000,C 90.000,E1 320.436} C_DIS
LIN {X 0.060,Y -614.069,Z 1072.574,A 0.000,B 0.000,C 90.000,E1 319.380} C_DIS
LIN {X -0.050,Y -613.246,Z 1072.566,A 0.000,B 0.000,C 90.000,E1 317.838} C_DIS
LIN {X 0.164,Y -612.409,Z 1072.560,A 0.000,B 0.000,C 90.000,E1 316.782} C_DIS
LIN {X 0.164,Y -611.505,Z 1072.553,A 0.000,B 0.000,C 90.000,E1 315.486} C_DIS
LIN {X 0.062,Y -610.075,Z 1072.541,A 0.000,B 0.000,C 90.000,E1 313.419} C_DIS
LIN {X -0.297,Y -609.542,Z 1072.538,A 0.000,B 0.000,C 90.000,E1 312.933} C_DIS
LIN {X 0.383,Y -609.500,Z 1072.537,A 0.000,B 0.000,C 90.000,E1 312.609} C_DIS
LIN {X 0.015,Y -608.988,Z 1072.534,A 0.000,B 0.000,C 90.000,E1 312.123} C_DIS
LIN {X 0.281,Y -608.967,Z 1072.533,A 0.000,B 0.000,C 90.000,E1 311.838} C_DIS
LIN {X -0.261,Y -607.191,Z 1072.521,A 0.000,B 0.000,C 90.000,E1 309.806} C_DIS
LIN {X -0.190,Y -606.717,Z 1072.518,A 0.000,B 0.000,C 90.000,E1 309.277} C_DIS
LIN {X 0.079,Y -606.645,Z 1072.517,A 0.000,B 0.000,C 90.000,E1 308.991} C_DIS
LIN {X -0.070,Y -605.243,Z 1072.505,A 0.000,B 0.000,C 90.000,E1 306.916} C_DIS
LIN {X 0.301,Y -604.028,Z 1072.496,A 0.000,B 0.000,C 90.000,E1 305.311} C_DIS
LIN {X 0.232,Y -603.235,Z 1072.492,A 0.000,B 0.000,C 90.000,E1 304.532} C_DIS
LIN {X -0.018,Y -602.125,Z 1072.485,A 0.000,B 0.000,C 90.000,E1 303.245} C_DIS
LIN {X 0.042,Y -600.757,Z 1072.477,A 0.000,B 0.000,C 90.000,E1 301.926} C_DIS
LIN {X 0.258,Y -598.675,Z 1072.470,A 0.000,B 0.000,C 90.000,E1 300.590} C_DIS
LIN {X 0.308,Y -596.740,Z 1072.466,A 0.000,B 0.000,C 90.000,E1 299.795} C_DIS
LIN {X 0.049,Y -594.582,Z 1072.461,A 0.000,B 0.000,C 90.000,E1 299.027} C_DIS
LIN {X 0.059,Y -591.863,Z 1072.457,A 0.000,B 0.000,C 90.000,E1 298.231} C_DIS
LIN {X -0.038,Y -590.823,Z 1072.455,A 0.000,B 0.000,C 90.000,E1 297.975} C_DIS
LIN {X 0.032,Y -588.312,Z 1072.453,A 0.000,B 0.000,C 90.000,E1 297.436} C_DIS
LIN {X -0.191,Y -585.751,Z 1072.449,A 0.000,B 0.000,C 90.000,E1 296.924} C_DIS
LIN {X 0.091,Y -582.458,Z 1072.447,A 0.000,B 0.000,C 90.000,E1 296.360} C_DIS
LIN {X -0.103,Y -579.635,Z 1072.444,A 0.000,B 0.000,C 90.000,E1 295.976} C_DIS
LIN {X -0.238,Y -577.339,Z 1072.443,A 0.000,B 0.000,C 90.000,E1 295.720} C_DIS
LIN {X 0.121,Y -573.763,Z 1072.441,A 0.000,B 0.000,C 90.000,E1 295.283} C_DIS
LIN {X 0.021,Y -569.336,Z 1072.438,A 0.000,B 0.000,C 90.000,E1 294.899} C_DIS
LIN {X 0.075,Y -567.007,Z 1072.438,A 0.000,B 0.000,C 90.000,E1 294.771} C_DIS
LIN {X 0.167,Y -561.406,Z 1072.436,A 0.000,B 0.000,C 90.000,E1 294.515} C_DIS
LIN {X 0.168,Y -556.739,Z 1072.436,A 0.000,B 0.000,C 90.000,E1 294.387} C_DIS
LIN {X 0.154,Y -554.549,Z 1072.435,A 0.000,B 0.000,C 90.000,E1 294.335} C_DIS
LIN {X 0.040,Y -552.258,Z 1072.435,A 0.000,B 0.000,C 90.000,E1 294.259} C_DIS
LIN {X -0.056,Y -547.298,Z 1072.432,A 0.000,B 0.000,C 90.000,E1 293.823} C_DIS
LIN {X -0.041,Y -546.159,Z 1072.432,A 0.000,B 0.000,C 90.000,E1 293.695} C_DIS
LIN {X -0.115,Y -545.484,Z 1072.431,A 0.000,B 0.000,C 90.000,E1 293.567} C_DIS
LIN {X 0.135,Y -544.793,Z 1072.429,A 0.000,B 0.000,C 90.000,E1 293.259} C_DIS
LIN {X 0.008,Y -544.250,Z 1072.429,A 0.000,B 0.000,C 90.000,E1 293.131} C_DIS
LIN {X -0.119,Y -543.976,Z 1072.428,A 0.000,B 0.000,C 90.000,E1 293.003} C_DIS
LIN {X -0.214,Y -543.747,Z 1072.425,A 0.000,B 0.000,C 90.000,E1 292.589} C_DIS
LIN {X 0.030,Y -543.346,Z 1072.424,A 0.000,B 0.000,C 90.000,E1 292.280} C_DIS
LIN {X 0.091,Y -542.930,Z 1072.421,A 0.000,B 0.000,C 90.000,E1 291.716} C_DIS
LIN {X 0.108,Y -542.887,Z 1072.403,A 0.000,B 0.000,C 90.000,E1 288.598} C_DIS
LIN {X -0.036,Y -543.010,Z 1072.394,A 0.000,B 0.000,C 90.000,E1 286.913} C_DIS
LIN {X 0.113,Y -542.748,Z 1072.386,A 0.000,B 0.000,C 90.000,E1 285.481} C_DIS
LIN {X 0.114,Y -542.280,Z 1072.378,A 0.000,B 0.000,C 90.000,E1 284.064} C_DIS
LIN {X 0.107,Y -541.757,Z 1072.370,A 0.000,B 0.000,C 90.000,E1 282.647} C_DIS
LIN {X 0.045,Y -540.873,Z 1072.361,A 0.000,B 0.000,C 90.000,E1 280.950} C_DIS
LIN {X -0.064,Y -539.783,Z 1072.350,A 0.000,B 0.000,C 90.000,E1 278.973} C_DIS
LIN {X 0.120,Y -538.985,Z 1072.342,A 0.000,B 0.000,C 90.000,E1 277.530} C_DIS
LIN {X -0.182,Y -538.056,Z 1072.333,A 0.000,B 0.000,C 90.000,E1 275.853} C_DIS
LIN {X -0.037,Y -536.996,Z 1072.321,A 0.000,B 0.000,C 90.000,E1 273.841} C_DIS
LIN {X 0.022,Y -535.963,Z 1072.310,A 0.000,B 0.000,C 90.000,E1 271.835} C_DIS
LIN {X 0.057,Y -535.007,Z 1072.301,A 0.000,B 0.000,C 90.000,E1 270.115} C_DIS
LIN {X 0.058,Y -534.188,Z 1072.293,A 0.000,B 0.000,C 90.000,E1 268.682} C_DIS
LIN {X 0.056,Y -533.365,Z 1072.285,A 0.000,B 0.000,C 90.000,E1 267.249} C_DIS
LIN {X 0.071,Y -532.496,Z 1072.277,A 0.000,B 0.000,C 90.000,E1 265.812} C_DIS
LIN {X 0.074,Y -531.443,Z 1072.269,A 0.000,B 0.000,C 90.000,E1 264.375} C_DIS
LIN {X 0.111,Y -530.156,Z 1072.261,A 0.000,B 0.000,C 90.000,E1 262.932} C_DIS
LIN {X 0.121,Y -528.675,Z 1072.253,A 0.000,B 0.000,C 90.000,E1 261.489} C_DIS
LIN {X 0.200,Y -526.811,Z 1072.243,A 0.000,B 0.000,C 90.000,E1 259.746} C_DIS
LIN {X -0.161,Y -524.648,Z 1072.232,A 0.000,B 0.000,C 90.000,E1 257.757} C_DIS
LIN {X 0.031,Y -523.140,Z 1072.224,A 0.000,B 0.000,C 90.000,E1 256.284} C_DIS
LIN {X -0.174,Y -521.092,Z 1072.213,A 0.000,B 0.000,C 90.000,E1 254.267} C_DIS
LIN {X 0.202,Y -518.940,Z 1072.201,A 0.000,B 0.000,C 90.000,E1 252.181} C_DIS
LIN {X -0.066,Y -517.695,Z 1072.195,A 0.000,B 0.000,C 90.000,E1 251.040} C_DIS
LIN {X 0.082,Y -515.707,Z 1072.185,A 0.000,B 0.000,C 90.000,E1 249.263} C_DIS
LIN {X 0.059,Y -513.745,Z 1072.177,A 0.000,B 0.000,C 90.000,E1 247.794} C_DIS
LIN {X 0.188,Y -511.709,Z 1072.169,A 0.000,B 0.000,C 90.000,E1 246.305} C_DIS
LIN {X 0.019,Y -509.471,Z 1072.160,A 0.000,B 0.000,C 90.000,E1 244.845} C_DIS
LIN {X -0.185,Y -507.098,Z 1072.152,A 0.000,B 0.000,C 90.000,E1 243.384} C_DIS
LIN {X 0.106,Y -504.102,Z 1072.142,A 0.000,B 0.000,C 90.000,E1 241.563} C_DIS
LIN {X 0.022,Y -501.528,Z 1072.134,A 0.000,B 0.000,C 90.000,E1 240.078} C_DIS
LIN {X -0.041,Y -498.861,Z 1072.125,A 0.000,B 0.000,C 90.000,E1 238.584} C_DIS
LIN {X 0.135,Y -495.544,Z 1072.115,A 0.000,B 0.000,C 90.000,E1 236.755} C_DIS
LIN {X -0.187,Y -491.988,Z 1072.105,A 0.000,B 0.000,C 90.000,E1 234.975} C_DIS
LIN {X -0.108,Y -489.496,Z 1072.099,A 0.000,B 0.000,C 90.000,E1 233.749} C_DIS
LIN {X 0.032,Y -486.951,Z 1072.092,A 0.000,B 0.000,C 90.000,E1 232.512} C_DIS
LIN {X -0.047,Y -484.220,Z 1072.085,A 0.000,B 0.000,C 90.000,E1 231.295} C_DIS
LIN {X -0.088,Y -481.552,Z 1072.078,A 0.000,B 0.000,C 90.000,E1 230.070} C_DIS
LIN {X 0.255,Y -476.251,Z 1072.064,A 0.000,B 0.000,C 90.000,E1 227.553} C_DIS
LIN {X 0.067,Y -471.450,Z 1072.051,A 0.000,B 0.000,C 90.000,E1 225.081} C_DIS
LIN {X -0.089,Y -468.009,Z 1072.040,A 0.000,B 0.000,C 90.000,E1 223.218} C_DIS
LIN {X -0.023,Y -464.973,Z 1072.031,A 0.000,B 0.000,C 90.000,E1 221.634} C_DIS
LIN {X 0.040,Y -461.116,Z 1072.021,A 0.000,B 0.000,C 90.000,E1 219.725} C_DIS
LIN {X -0.029,Y -458.005,Z 1072.012,A 0.000,B 0.000,C 90.000,E1 218.141} C_DIS
LIN {X 0.001,Y -454.837,Z 1072.003,A 0.000,B 0.000,C 90.000,E1 216.537} C_DIS
LIN {X 0.048,Y -450.153,Z 1071.990,A 0.000,B 0.000,C 90.000,E1 214.278} C_DIS
LIN {X 0.076,Y -445.652,Z 1071.978,A 0.000,B 0.000,C 90.000,E1 212.005} C_DIS
LIN {X -0.051,Y -443.219,Z 1071.971,A 0.000,B 0.000,C 90.000,E1 210.718} C_DIS
LIN {X -0.015,Y -440.051,Z 1071.962,A 0.000,B 0.000,C 90.000,E1 209.077} C_DIS
LIN {X 0.021,Y -435.120,Z 1071.947,A 0.000,B 0.000,C 90.000,E1 206.437} C_DIS
LIN {X 0.083,Y -432.817,Z 1071.940,A 0.000,B 0.000,C 90.000,E1 205.103} C_DIS
LIN {X 0.107,Y -429.026,Z 1071.927,A 0.000,B 0.000,C 90.000,E1 202.770} C_DIS
LIN {X 0.085,Y -425.811,Z 1071.914,A 0.000,B 0.000,C 90.000,E1 200.429} C_DIS
LIN {X 0.061,Y -424.681,Z 1071.906,A 0.000,B 0.000,C 90.000,E1 199.087} C_DIS
LIN {X 0.041,Y -424.362,Z 1071.902,A 0.000,B 0.000,C 90.000,E1 198.417} C_DIS
LIN {X -0.114,Y -424.372,Z 1071.899,A 0.000,B 0.000,C 90.000,E1 197.764} C_DIS
LIN {X -0.141,Y -424.773,Z 1071.895,A 0.000,B 0.000,C 90.000,E1 197.094} C_DIS
LIN {X 0.116,Y -425.575,Z 1071.891,A 0.000,B 0.000,C 90.000,E1 196.386} C_DIS
LIN {X -0.102,Y -426.135,Z 1071.889,A 0.000,B 0.000,C 90.000,E1 196.079} C_DIS
LIN {X 0.170,Y -427.698,Z 1071.886,A 0.000,B 0.000,C 90.000,E1 195.371} C_DIS
LIN {X 0.246,Y -430.867,Z 1071.880,A 0.000,B 0.000,C 90.000,E1 194.356} C_DIS
LIN {X -0.154,Y -435.851,Z 1071.874,A 0.000,B 0.000,C 90.000,E1 193.244} C_DIS
LIN {X -0.106,Y -439.723,Z 1071.869,A 0.000,B 0.000,C 90.000,E1 192.411} C_DIS
LIN {X -0.038,Y -449.308,Z 1071.859,A 0.000,B 0.000,C 90.000,E1 190.602} C_DIS
LIN {X 0.036,Y -462.276,Z 1071.846,A 0.000,B 0.000,C 90.000,E1 188.341} C_DIS
LIN {X 0.249,Y -470.655,Z 1071.839,A 0.000,B 0.000,C 90.000,E1 186.891} C_DIS
LIN {X 0.117,Y -476.033,Z 1071.833,A 0.000,B 0.000,C 90.000,E1 185.967} C_DIS
LIN {X -0.163,Y -482.886,Z 1071.826,A 0.000,B 0.000,C 90.000,E1 184.759} C_DIS
LIN {X -0.051,Y -488.822,Z 1071.820,A 0.000,B 0.000,C 90.000,E1 183.669} C_DIS
LIN {X 0.146,Y -494.625,Z 1071.814,A 0.000,B 0.000,C 90.000,E1 182.579} C_DIS
LIN {X -0.077,Y -500.330,Z 1071.809,A 0.000,B 0.000,C 90.000,E1 181.547} C_DIS
LIN {X 0.156,Y -507.432,Z 1071.801,A 0.000,B 0.000,C 90.000,E1 180.172} C_DIS
LIN {X 0.222,Y -515.300,Z 1071.793,A 0.000,B 0.000,C 90.000,E1 178.682} C_DIS
LIN {X -0.253,Y -520.755,Z 1071.787,A 0.000,B 0.000,C 90.000,E1 177.707} C_DIS
LIN {X -0.211,Y -529.114,Z 1071.778,A 0.000,B 0.000,C 90.000,E1 176.102} C_DIS
LIN {X 0.080,Y -537.392,Z 1071.770,A 0.000,B 0.000,C 90.000,E1 174.489} C_DIS
LIN {X 0.211,Y -544.844,Z 1071.762,A 0.000,B 0.000,C 90.000,E1 173.053} C_DIS
LIN {X 0.245,Y -551.443,Z 1071.755,A 0.000,B 0.000,C 90.000,E1 171.781} C_DIS
LIN {X -0.075,Y -557.875,Z 1071.748,A 0.000,B 0.000,C 90.000,E1 170.557} C_DIS
LIN {X 0.019,Y -564.781,Z 1071.740,A 0.000,B 0.000,C 90.000,E1 169.162} C_DIS
LIN {X 0.156,Y -570.180,Z 1071.734,A 0.000,B 0.000,C 90.000,E1 168.049} C_DIS
LIN {X -0.191,Y -575.249,Z 1071.728,A 0.000,B 0.000,C 90.000,E1 166.992} C_DIS
LIN {X -0.012,Y -580.870,Z 1071.721,A 0.000,B 0.000,C 90.000,E1 165.755} C_DIS
LIN {X 0.159,Y -586.756,Z 1071.713,A 0.000,B 0.000,C 90.000,E1 164.393} C_DIS
LIN {X 0.169,Y -591.161,Z 1071.708,A 0.000,B 0.000,C 90.000,E1 163.323} C_DIS
LIN {X -0.028,Y -594.286,Z 1071.703,A 0.000,B 0.000,C 90.000,E1 162.543} C_DIS
LIN {X 0.259,Y -598.288,Z 1071.697,A 0.000,B 0.000,C 90.000,E1 161.456} C_DIS
LIN {X 0.038,Y -602.011,Z 1071.691,A 0.000,B 0.000,C 90.000,E1 160.423} C_DIS
LIN {X -0.135,Y -605.566,Z 1071.685,A 0.000,B 0.000,C 90.000,E1 159.390} C_DIS
LIN {X 0.185,Y -610.476,Z 1071.677,A 0.000,B 0.000,C 90.000,E1 157.794} C_DIS
LIN {X -0.185,Y -612.817,Z 1071.672,A 0.000,B 0.000,C 90.000,E1 157.050} C_DIS
LIN {X -0.027,Y -616.432,Z 1071.665,A 0.000,B 0.000,C 90.000,E1 155.741} C_DIS
LIN {X -0.110,Y -619.929,Z 1071.658,A 0.000,B 0.000,C 90.000,E1 154.460} C_DIS
LIN {X -0.121,Y -623.755,Z 1071.650,A 0.000,B 0.000,C 90.000,E1 152.922} C_DIS
LIN {X -0.089,Y -626.324,Z 1071.644,A 0.000,B 0.000,C 90.000,E1 151.897} C_DIS
LIN {X 0.294,Y -629.331,Z 1071.637,A 0.000,B 0.000,C 90.000,E1 150.589} C_DIS
LIN {X 0.180,Y -632.232,Z 1071.630,A 0.000,B 0.000,C 90.000,E1 149.331} C_DIS
LIN {X -0.032,Y -636.069,Z 1071.620,A 0.000,B 0.000,C 90.000,E1 147.582} C_DIS
LIN {X 0.183,Y -639.725,Z 1071.610,A 0.000,B 0.000,C 90.000,E1 145.801} C_DIS
LIN {X 0.028,Y -642.287,Z 1071.603,A 0.000,B 0.000,C 90.000,E1 144.562} C_DIS
LIN {X 0.182,Y -645.284,Z 1071.595,A 0.000,B 0.000,C 90.000,E1 143.050} C_DIS
LIN {X -0.025,Y -647.795,Z 1071.588,A 0.000,B 0.000,C 90.000,E1 141.823} C_DIS
LIN {X -0.201,Y -650.269,Z 1071.581,A 0.000,B 0.000,C 90.000,E1 140.598} C_DIS
LIN {X 0.012,Y -653.319,Z 1071.573,A 0.000,B 0.000,C 90.000,E1 139.094} C_DIS
LIN {X -0.205,Y -656.458,Z 1071.565,A 0.000,B 0.000,C 90.000,E1 137.634} C_DIS
LIN {X 0.022,Y -661.318,Z 1071.552,A 0.000,B 0.000,C 90.000,E1 135.405} C_DIS
LIN {X -0.057,Y -664.929,Z 1071.544,A 0.000,B 0.000,C 90.000,E1 133.947} C_DIS
LIN {X -0.036,Y -669.369,Z 1071.535,A 0.000,B 0.000,C 90.000,E1 132.243} C_DIS
LIN {X 0.074,Y -673.094,Z 1071.527,A 0.000,B 0.000,C 90.000,E1 130.782} C_DIS
LIN {X 0.226,Y -676.304,Z 1071.520,A 0.000,B 0.000,C 90.000,E1 129.564} C_DIS
LIN {X 0.171,Y -681.161,Z 1071.509,A 0.000,B 0.000,C 90.000,E1 127.649} C_DIS
LIN {X -0.024,Y -683.669,Z 1071.504,A 0.000,B 0.000,C 90.000,E1 126.710} C_DIS
LIN {X 0.364,Y -686.165,Z 1071.499,A 0.000,B 0.000,C 90.000,E1 125.724} C_DIS
LIN {X 0.051,Y -689.580,Z 1071.491,A 0.000,B 0.000,C 90.000,E1 124.326} C_DIS
LIN {X -0.227,Y -692.474,Z 1071.484,A 0.000,B 0.000,C 90.000,E1 123.166} C_DIS
LIN {X 0.131,Y -695.320,Z 1071.478,A 0.000,B 0.000,C 90.000,E1 121.957} C_DIS
LIN {X -0.056,Y -697.954,Z 1071.471,A 0.000,B 0.000,C 90.000,E1 120.797} C_DIS
LIN {X 0.115,Y -699.493,Z 1071.467,A 0.000,B 0.000,C 90.000,E1 120.079} C_DIS
LIN {X -0.304,Y -700.638,Z 1071.463,A 0.000,B 0.000,C 90.000,E1 119.411} C_DIS
LIN {X -0.104,Y -701.504,Z 1071.459,A 0.000,B 0.000,C 90.000,E1 118.693} C_DIS
LIN {X 0.220,Y -703.484,Z 1071.448,A 0.000,B 0.000,C 90.000,E1 116.565} C_DIS
LIN {X -0.191,Y -704.221,Z 1071.444,A 0.000,B 0.000,C 90.000,E1 115.899} C_DIS
LIN {X 0.009,Y -704.852,Z 1071.439,A 0.000,B 0.000,C 90.000,E1 114.951} C_DIS
LIN {X 0.001,Y -704.940,Z 1071.437,A 0.000,B 0.000,C 90.000,E1 114.719} C_DIS
LIN {X -0.068,Y -704.618,Z 1071.435,A 0.000,B 0.000,C 90.000,E1 114.259} C_DIS
LIN {X -0.070,Y -704.371,Z 1071.433,A 0.000,B 0.000,C 90.000,E1 114.027} C_DIS
LIN {X -0.147,Y -702.929,Z 1071.431,A 0.000,B 0.000,C 90.000,E1 113.567} C_DIS
LIN {X -0.147,Y -702.036,Z 1071.430,A 0.000,B 0.000,C 90.000,E1 113.334} C_DIS
LIN {X 0.125,Y -698.581,Z 1071.427,A 0.000,B 0.000,C 90.000,E1 112.845} C_DIS
LIN {X -0.387,Y -697.620,Z 1071.426,A 0.000,B 0.000,C 90.000,E1 112.770} C_DIS
LIN {X -0.255,Y -696.232,Z 1071.426,A 0.000,B 0.000,C 90.000,E1 112.642} C_DIS
LIN {X -0.021,Y -694.195,Z 1071.425,A 0.000,B 0.000,C 90.000,E1 112.514} C_DIS
LIN {X -0.262,Y -686.868,Z 1071.423,A 0.000,B 0.000,C 90.000,E1 112.206} C_DIS
LIN {X 0.125,Y -684.269,Z 1071.423,A 0.000,B 0.000,C 90.000,E1 112.099} C_DIS
LIN {X -0.228,Y -675.824,Z 1071.422,A 0.000,B 0.000,C 90.000,E1 112.025} C_DIS
LIN {X -0.261,Y -607.315,Z 1071.422,A 0.000,B 0.000,C 90.000,E1 112.025} C_DIS
LIN {X -0.039,Y -603.385,Z 1071.421,A 0.000,B 0.000,C 90.000,E1 111.844} C_DIS
LIN {X 0.143,Y -599.002,Z 1071.420,A 0.000,B 0.000,C 90.000,E1 111.589} C_DIS
LIN {X 0.141,Y -596.078,Z 1071.419,A 0.000,B 0.000,C 90.000,E1 111.408} C_DIS
LIN {X -0.028,Y -588.862,Z 1071.416,A 0.000,B 0.000,C 90.000,E1 110.865} C_DIS
LIN {X -0.124,Y -580.493,Z 1071.412,A 0.000,B 0.000,C 90.000,E1 110.174} C_DIS
LIN {X 0.180,Y -575.223,Z 1071.410,A 0.000,B 0.000,C 90.000,E1 109.704} C_DIS
LIN {X 0.065,Y -569.190,Z 1071.407,A 0.000,B 0.000,C 90.000,E1 109.268} C_DIS
LIN {X -0.141,Y -560.883,Z 1071.404,A 0.000,B 0.000,C 90.000,E1 108.779} C_DIS
LIN {X -0.187,Y -554.334,Z 1071.402,A 0.000,B 0.000,C 90.000,E1 108.417} C_DIS
LIN {X -0.054,Y -549.320,Z 1071.400,A 0.000,B 0.000,C 90.000,E1 108.055} C_DIS
LIN {X -0.190,Y -547.690,Z 1071.399,A 0.000,B 0.000,C 90.000,E1 107.873} C_DIS
LIN {X -0.232,Y -547.666,Z 1071.399,A 0.000,B 0.000,C 90.000,E1 107.873} C_DIS
LIN {X -0.204,Y -547.348,Z 1071.398,A 0.000,B 0.000,C 90.000,E1 107.638} C_DIS
LIN {X -0.306,Y -547.608,Z 1071.393,A 0.000,B 0.000,C 90.000,E1 106.804} C_DIS
LIN {X -0.157,Y -548.388,Z 1071.387,A 0.000,B 0.000,C 90.000,E1 105.662} C_DIS
LIN {X -0.133,Y -549.966,Z 1071.375,A 0.000,B 0.000,C 90.000,E1 103.411} C_DIS
LIN {X 0.228,Y -551.898,Z 1071.362,A 0.000,B 0.000,C 90.000,E1 101.130} C_DIS
LIN {X 0.004,Y -554.262,Z 1071.350,A 0.000,B 0.000,C 90.000,E1 98.916} C_DIS
LIN {X 0.042,Y -556.149,Z 1071.340,A 0.000,B 0.000,C 90.000,E1 97.239} C_DIS
LIN {X -0.011,Y -557.721,Z 1071.333,A 0.000,B 0.000,C 90.000,E1 95.853} C_DIS
LIN {X -0.097,Y -559.048,Z 1071.325,A 0.000,B 0.000,C 90.000,E1 94.473} C_DIS
LIN {X -0.165,Y -559.912,Z 1071.317,A 0.000,B 0.000,C 90.000,E1 93.094} C_DIS
LIN {X -0.252,Y -560.647,Z 1071.309,A 0.000,B 0.000,C 90.000,E1 91.718} C_DIS
LIN {X -0.241,Y -561.405,Z 1071.300,A 0.000,B 0.000,C 90.000,E1 90.057} C_DIS
LIN {X 0.249,Y -561.878,Z 1071.293,A 0.000,B 0.000,C 90.000,E1 88.625} C_DIS
LIN {X -0.137,Y -562.661,Z 1071.282,A 0.000,B 0.000,C 90.000,E1 86.731} C_DIS
LIN {X -0.176,Y -563.174,Z 1071.274,A 0.000,B 0.000,C 90.000,E1 85.355} C_DIS
LIN {X -0.023,Y -563.697,Z 1071.265,A 0.000,B 0.000,C 90.000,E1 83.685} C_DIS
LIN {X 0.213,Y -564.167,Z 1071.256,A 0.000,B 0.000,C 90.000,E1 82.008} C_DIS
LIN {X 0.231,Y -564.918,Z 1071.244,A 0.000,B 0.000,C 90.000,E1 79.803} C_DIS
LIN {X 0.190,Y -565.764,Z 1071.233,A 0.000,B 0.000,C 90.000,E1 77.881} C_DIS
LIN {X -0.144,Y -566.816,Z 1071.222,A 0.000,B 0.000,C 90.000,E1 75.992} C_DIS
LIN {X -0.003,Y -568.922,Z 1071.205,A 0.000,B 0.000,C 90.000,E1 72.960} C_DIS
LIN {X 0.051,Y -570.438,Z 1071.195,A 0.000,B 0.000,C 90.000,E1 71.040} C_DIS
LIN {X 0.160,Y -571.828,Z 1071.186,A 0.000,B 0.000,C 90.000,E1 69.390} C_DIS
LIN {X -0.237,Y -573.146,Z 1071.177,A 0.000,B 0.000,C 90.000,E1 67.794} C_DIS
LIN {X 0.158,Y -574.002,Z 1071.171,A 0.000,B 0.000,C 90.000,E1 66.666} C_DIS
LIN {X 0.174,Y -575.043,Z 1071.163,A 0.000,B 0.000,C 90.000,E1 65.305} C_DIS
LIN {X 0.019,Y -576.048,Z 1071.154,A 0.000,B 0.000,C 90.000,E1 63.691} C_DIS
LIN {X -0.099,Y -576.938,Z 1071.145,A 0.000,B 0.000,C 90.000,E1 62.076} C_DIS
LIN {X -0.056,Y -577.722,Z 1071.137,A 0.000,B 0.000,C 90.000,E1 60.717} C_DIS
LIN {X 0.277,Y -578.369,Z 1071.130,A 0.000,B 0.000,C 90.000,E1 59.331} C_DIS
LIN {X 0.120,Y -578.953,Z 1071.122,A 0.000,B 0.000,C 90.000,E1 57.995} C_DIS
LIN {X 0.279,Y -579.563,Z 1071.115,A 0.000,B 0.000,C 90.000,E1 56.628} C_DIS
LIN {X -0.196,Y -580.008,Z 1071.109,A 0.000,B 0.000,C 90.000,E1 55.595} C_DIS
LIN {X 0.139,Y -580.412,Z 1071.103,A 0.000,B 0.000,C 90.000,E1 54.482} C_DIS
LIN {X 0.005,Y -580.666,Z 1071.097,A 0.000,B 0.000,C 90.000,E1 53.417} C_DIS
LIN {X -0.128,Y -580.822,Z 1071.091,A 0.000,B 0.000,C 90.000,E1 52.351} C_DIS
LIN {X -0.075,Y -580.764,Z 1071.086,A 0.000,B 0.000,C 90.000,E1 51.537} C_DIS
LIN {X -0.019,Y -580.660,Z 1071.082,A 0.000,B 0.000,C 90.000,E1 50.723} C_DIS
LIN {X 0.084,Y -580.093,Z 1071.073,A 0.000,B 0.000,C 90.000,E1 49.094} C_DIS
LIN {X -0.042,Y -579.499,Z 1071.065,A 0.000,B 0.000,C 90.000,E1 47.757} C_DIS
LIN {X 0.254,Y -578.685,Z 1071.058,A 0.000,B 0.000,C 90.000,E1 46.377} C_DIS
LIN {X -0.032,Y -577.867,Z 1071.052,A 0.000,B 0.000,C 90.000,E1 45.324} C_DIS
LIN {X -0.046,Y -577.083,Z 1071.047,A 0.000,B 0.000,C 90.000,E1 44.514} C_DIS
LIN {X 0.063,Y -575.710,Z 1071.041,A 0.000,B 0.000,C 90.000,E1 43.419} C_DIS
LIN {X -0.267,Y -574.182,Z 1071.035,A 0.000,B 0.000,C 90.000,E1 42.366} C_DIS
LIN {X 0.226,Y -572.535,Z 1071.029,A 0.000,B 0.000,C 90.000,E1 41.229} C_DIS
LIN {X -0.110,Y -570.415,Z 1071.023,A 0.000,B 0.000,C 90.000,E1 40.172} C_DIS
LIN {X -0.036,Y -567.925,Z 1071.017,A 0.000,B 0.000,C 90.000,E1 39.072} C_DIS
LIN {X 0.006,Y -565.151,Z 1071.011,A 0.000,B 0.000,C 90.000,E1 37.971} C_DIS
LIN {X -0.104,Y -562.719,Z 1071.006,A 0.000,B 0.000,C 90.000,E1 37.156} C_DIS
LIN {X 0.105,Y -560.916,Z 1071.003,A 0.000,B 0.000,C 90.000,E1 36.583} C_DIS
LIN {X 0.064,Y -557.785,Z 1070.999,A 0.000,B 0.000,C 90.000,E1 35.758} C_DIS
LIN {X -0.216,Y -555.639,Z 1070.996,A 0.000,B 0.000,C 90.000,E1 35.231} C_DIS
LIN {X -0.119,Y -551.389,Z 1070.990,A 0.000,B 0.000,C 90.000,E1 34.246} C_DIS
LIN {X 0.194,Y -547.381,Z 1070.986,A 0.000,B 0.000,C 90.000,E1 33.372} C_DIS
LIN {X 0.142,Y -543.762,Z 1070.982,A 0.000,B 0.000,C 90.000,E1 32.673} C_DIS
LIN {X 0.234,Y -538.509,Z 1070.976,A 0.000,B 0.000,C 90.000,E1 31.671} C_DIS
LIN {X -0.043,Y -535.287,Z 1070.973,A 0.000,B 0.000,C 90.000,E1 31.131} C_DIS
LIN {X 0.118,Y -531.822,Z 1070.970,A 0.000,B 0.000,C 90.000,E1 30.541} C_DIS
LIN {X -0.204,Y -528.127,Z 1070.967,A 0.000,B 0.000,C 90.000,E1 30.001} C_DIS
LIN {X -0.094,Y -524.163,Z 1070.963,A 0.000,B 0.000,C 90.000,E1 29.411} C_DIS
LIN {X -0.174,Y -518.831,Z 1070.959,A 0.000,B 0.000,C 90.000,E1 28.693} C_DIS
LIN {X 0.034,Y -515.447,Z 1070.957,A 0.000,B 0.000,C 90.000,E1 28.231} C_DIS
LIN {X 0.221,Y -511.851,Z 1070.954,A 0.000,B 0.000,C 90.000,E1 27.769} C_DIS
LIN {X -0.132,Y -504.188,Z 1070.950,A 0.000,B 0.000,C 90.000,E1 26.924} C_DIS
LIN {X 0.060,Y -497.429,Z 1070.946,A 0.000,B 0.000,C 90.000,E1 26.181} C_DIS
LIN {X -0.065,Y -487.812,Z 1070.940,A 0.000,B 0.000,C 90.000,E1 25.207} C_DIS
LIN {X 0.195,Y -477.728,Z 1070.935,A 0.000,B 0.000,C 90.000,E1 24.207} C_DIS
LIN {X -0.127,Y -468.841,Z 1070.930,A 0.000,B 0.000,C 90.000,E1 23.439} C_DIS
LIN {X -0.001,Y -462.801,Z 1070.927,A 0.000,B 0.000,C 90.000,E1 22.898} C_DIS
LIN {X 0.157,Y -449.389,Z 1070.921,A 0.000,B 0.000,C 90.000,E1 21.716} C_DIS
LIN {X 0.113,Y -431.754,Z 1070.912,A 0.000,B 0.000,C 90.000,E1 20.120} C_DIS
LIN {X -0.123,Y -418.894,Z 1070.905,A 0.000,B 0.000,C 90.000,E1 18.852} C_DIS
LIN {X -0.077,Y -410.599,Z 1070.900,A 0.000,B 0.000,C 90.000,E1 17.928} C_DIS
LIN {X -0.223,Y -401.234,Z 1070.893,A 0.000,B 0.000,C 90.000,E1 16.804} C_DIS
LIN {X -0.132,Y -397.849,Z 1070.891,A 0.000,B 0.000,C 90.000,E1 16.315} C_DIS
LIN {X -0.093,Y -393.987,Z 1070.887,A 0.000,B 0.000,C 90.000,E1 15.607} C_DIS
LIN {X -0.035,Y -392.779,Z 1070.885,A 0.000,B 0.000,C 90.000,E1 15.245} C_DIS
LIN {X -0.038,Y -391.889,Z 1070.881,A 0.000,B 0.000,C 90.000,E1 14.537} C_DIS
LIN {X -0.048,Y -391.991,Z 1070.877,A 0.000,B 0.000,C 90.000,E1 13.828} C_DIS
LIN {X -0.087,Y -393.374,Z 1070.870,A 0.000,B 0.000,C 90.000,E1 12.591} C_DIS
LIN {X 0.018,Y -400.231,Z 1070.846,A 0.000,B 0.000,C 90.000,E1 8.341} C_DIS
LIN {X -0.091,Y -405.382,Z 1070.833,A 0.000,B 0.000,C 90.000,E1 5.910} C_DIS
LIN {X -0.166,Y -408.884,Z 1070.824,A 0.000,B 0.000,C 90.000,E1 4.359} C_DIS
LIN {X -0.177,Y -409.352,Z 1070.823,A 0.000,B 0.000,C 90.000,E1 4.188} C_DIS
LIN {X -0.023,Y -411.795,Z 1070.820,A 0.000,B 0.000,C 90.000,E1 3.555} C_DIS
LIN {X 0.135,Y -417.056,Z 1070.816,A 0.000,B 0.000,C 90.000,E1 2.808} C_DIS
LIN {X 0.094,Y -419.106,Z 1070.815,A 0.000,B 0.000,C 90.000,E1 2.636} C_DIS
LIN {X 0.143,Y -423.736,Z 1070.813,A 0.000,B 0.000,C 90.000,E1 2.293} C_DIS
LIN {X -0.016,Y -437.134,Z 1070.808,A 0.000,B 0.000,C 90.000,E1 1.432} C_DIS
LIN {X 0.000,Y -459.659,Z 1070.800,A 0.000,B 0.000,C 90.000,E1 360.000} C_DIS
LIN {X 0.069,Y -476.221,Z 1070.794,A 0.000,B 0.000,C 90.000,E1 358.969} C_DIS
LIN {X -0.065,Y -485.708,Z 1070.791,A 0.000,B 0.000,C 90.000,E1 358.396} C_DIS
LIN {X -0.069,Y -493.751,Z 1070.788,A 0.000,B 0.000,C 90.000,E1 357.879} C_DIS
LIN {X -0.214,Y -501.655,Z 1070.785,A 0.000,B 0.000,C 90.000,E1 357.364} C_DIS
LIN {X 0.192,Y -509.241,Z 1070.782,A 0.000,B 0.000,C 90.000,E1 356.788} C_DIS
LIN {X -0.251,Y -516.623,Z 1070.779,A 0.000,B 0.000,C 90.000,E1 356.274} C_DIS
LIN {X 0.094,Y -523.833,Z 1070.776,A 0.000,B 0.000,C 90.000,E1 355.641} C_DIS
LIN {X -0.104,Y -532.039,Z 1070.772,A 0.000,B 0.000,C 90.000,E1 354.894} C_DIS
LIN {X -0.232,Y -537.306,Z 1070.769,A 0.000,B 0.000,C 90.000,E1 354.375} C_DIS
LIN {X -0.250,Y -544.451,Z 1070.764,A 0.000,B 0.000,C 90.000,E1 353.571} C_DIS
LIN {X 0.114,Y -547.982,Z 1070.762,A 0.000,B 0.000,C 90.000,E1 353.109} C_DIS
LIN {X 0.053,Y -553.106,Z 1070.758,A 0.000,B 0.000,C 90.000,E1 352.413} C_DIS
LIN {X -0.040,Y -557.716,Z 1070.754,A 0.000,B 0.000,C 90.000,E1 351.724} C_DIS
LIN {X 0.234,Y -561.033,Z 1070.751,A 0.000,B 0.000,C 90.000,E1 351.141} C_DIS
LIN {X 0.295,Y -564.842,Z 1070.747,A 0.000,B 0.000,C 90.000,E1 350.443} C_DIS
LIN {X 0.147,Y -568.928,Z 1070.743,A 0.000,B 0.000,C 90.000,E1 349.634} C_DIS
LIN {X 0.095,Y -574.415,Z 1070.736,A 0.000,B 0.000,C 90.000,E1 348.409} C_DIS
LIN {X 0.145,Y -577.815,Z 1070.731,A 0.000,B 0.000,C 90.000,E1 347.589} C_DIS
LIN {X 0.018,Y -582.056,Z 1070.725,A 0.000,B 0.000,C 90.000,E1 346.520} C_DIS
LIN {X 0.148,Y -585.053,Z 1070.721,A 0.000,B 0.000,C 90.000,E1 345.700} C_DIS
LIN {X 0.133,Y -588.844,Z 1070.715,A 0.000,B 0.000,C 90.000,E1 344.629} C_DIS
LIN {X 0.172,Y -592.514,Z 1070.709,A 0.000,B 0.000,C 90.000,E1 343.559} C_DIS
LIN {X -0.313,Y -596.049,Z 1070.703,A 0.000,B 0.000,C 90.000,E1 342.543} C_DIS
LIN {X 0.105,Y -598.534,Z 1070.698,A 0.000,B 0.000,C 90.000,E1 341.710} C_DIS
LIN {X -0.121,Y -601.637,Z 1070.693,A 0.000,B 0.000,C 90.000,E1 340.678} C_DIS
LIN {X -0.097,Y -604.511,Z 1070.687,A 0.000,B 0.000,C 90.000,E1 339.625} C_DIS
LIN {X -0.175,Y -606.491,Z 1070.682,A 0.000,B 0.000,C 90.000,E1 338.847} C_DIS
LIN {X -0.078,Y -608.960,Z 1070.677,A 0.000,B 0.000,C 90.000,E1 337.794} C_DIS
LIN {X 0.099,Y -610.567,Z 1070.672,A 0.000,B 0.000,C 90.000,E1 336.997} C_DIS
LIN {X -0.063,Y -612.553,Z 1070.667,A 0.000,B 0.000,C 90.000,E1 335.973} C_DIS
LIN {X 0.113,Y -614.243,Z 1070.661,A 0.000,B 0.000,C 90.000,E1 334.921} C_DIS
LIN {X -0.030,Y -616.409,Z 1070.652,A 0.000,B 0.000,C 90.000,E1 333.384} C_DIS
LIN {X -0.084,Y -617.285,Z 1070.648,A 0.000,B 0.000,C 90.000,E1 332.615} C_DIS
LIN {X -0.132,Y -618.187,Z 1070.644,A 0.000,B 0.000,C 90.000,E1 331.847} C_DIS
LIN {X 0.095,Y -619.279,Z 1070.636,A 0.000,B 0.000,C 90.000,E1 330.539} C_DIS
LIN {X -0.173,Y -619.756,Z 1070.632,A 0.000,B 0.000,C 90.000,E1 329.793} C_DIS
LIN {X 0.090,Y -620.158,Z 1070.626,A 0.000,B 0.000,C 90.000,E1 328.742} C_DIS
LIN {X 0.150,Y -620.245,Z 1070.621,A 0.000,B 0.000,C 90.000,E1 327.709} C_DIS
LIN {X -0.120,Y -620.031,Z 1070.615,A 0.000,B 0.000,C 90.000,E1 326.707} C_DIS
LIN {X -0.059,Y -619.539,Z 1070.609,A 0.000,B 0.000,C 90.000,E1 325.674} C_DIS
LIN {X -0.010,Y -618.867,Z 1070.604,A 0.000,B 0.000,C 90.000,E1 324.642} C_DIS
LIN {X -0.035,Y -617.575,Z 1070.594,A 0.000,B 0.000,C 90.000,E1 322.844} C_DIS
LIN {X -0.008,Y -616.587,Z 1070.585,A 0.000,B 0.000,C 90.000,E1 321.295} C_DIS
LIN {X 0.044,Y -616.042,Z 1070.581,A 0.000,B 0.000,C 90.000,E1 320.517} C_DIS
LIN {X 0.303,Y -615.636,Z 1070.575,A 0.000,B 0.000,C 90.000,E1 319.461} C_DIS
LIN {X -0.034,Y -615.295,Z 1070.572,A 0.000,B 0.000,C 90.000,E1 318.976} C_DIS
LIN {X 0.263,Y -615.245,Z 1070.571,A 0.000,B 0.000,C 90.000,E1 318.690} C_DIS
LIN {X 0.389,Y -614.913,Z 1070.568,A 0.000,B 0.000,C 90.000,E1 318.162} C_DIS
LIN {X 0.222,Y -614.888,Z 1070.566,A 0.000,B 0.000,C 90.000,E1 317.919} C_DIS
LIN {X -0.045,Y -613.684,Z 1070.556,A 0.000,B 0.000,C 90.000,E1 316.134} C_DIS
LIN {X -0.018,Y -612.893,Z 1070.549,A 0.000,B 0.000,C 90.000,E1 314.838} C_DIS
LIN {X -0.181,Y -611.927,Z 1070.541,A 0.000,B 0.000,C 90.000,E1 313.299} C_DIS
LIN {X -0.260,Y -611.416,Z 1070.536,A 0.000,B 0.000,C 90.000,E1 312.528} C_DIS
LIN {X 0.015,Y -611.172,Z 1070.535,A 0.000,B 0.000,C 90.000,E1 312.243} C_DIS
LIN {X -0.341,Y -610.948,Z 1070.532,A 0.000,B 0.000,C 90.000,E1 311.757} C_DIS
LIN {X 0.029,Y -609.373,Z 1070.520,A 0.000,B 0.000,C 90.000,E1 309.644} C_DIS
LIN {X -0.111,Y -608.495,Z 1070.512,A 0.000,B 0.000,C 90.000,E1 308.096} C_DIS
LIN {X -0.098,Y -607.248,Z 1070.500,A 0.000,B 0.000,C 90.000,E1 306.011} C_DIS
LIN {X 0.136,Y -606.468,Z 1070.494,A 0.000,B 0.000,C 90.000,E1 304.945} C_DIS
LIN {X -0.063,Y -605.592,Z 1070.487,A 0.000,B 0.000,C 90.000,E1 303.658} C_DIS
LIN {X -0.192,Y -604.881,Z 1070.481,A 0.000,B 0.000,C 90.000,E1 302.625} C_DIS
LIN {X 0.245,Y -604.251,Z 1070.477,A 0.000,B 0.000,C 90.000,E1 301.799} C_DIS
LIN {X 0.008,Y -602.770,Z 1070.470,A 0.000,B 0.000,C 90.000,E1 300.512} C_DIS
LIN {X -0.130,Y -602.020,Z 1070.467,A 0.000,B 0.000,C 90.000,E1 300.001} C_DIS
LIN {X -0.198,Y -601.403,Z 1070.465,A 0.000,B 0.000,C 90.000,E1 299.745} C_DIS
LIN {X 0.029,Y -601.009,Z 1070.464,A 0.000,B 0.000,C 90.000,E1 299.461} C_DIS
LIN {X -0.187,Y -599.386,Z 1070.459,A 0.000,B 0.000,C 90.000,E1 298.693} C_DIS
LIN {X -0.131,Y -597.089,Z 1070.455,A 0.000,B 0.000,C 90.000,E1 297.897} C_DIS
LIN {X -0.211,Y -596.240,Z 1070.453,A 0.000,B 0.000,C 90.000,E1 297.641} C_DIS
LIN {X -0.292,Y -595.136,Z 1070.452,A 0.000,B 0.000,C 90.000,E1 297.385} C_DIS
LIN {X 0.152,Y -594.366,Z 1070.451,A 0.000,B 0.000,C 90.000,E1 297.078} C_DIS
LIN {X -0.072,Y -591.731,Z 1070.447,A 0.000,B 0.000,C 90.000,E1 296.437} C_DIS
LIN {X -0.010,Y -589.043,Z 1070.444,A 0.000,B 0.000,C 90.000,E1 295.899} C_DIS
LIN {X 0.299,Y -585.865,Z 1070.441,A 0.000,B 0.000,C 90.000,E1 295.335} C_DIS
LIN {X 0.120,Y -583.144,Z 1070.439,A 0.000,B 0.000,C 90.000,E1 294.951} C_DIS
LIN {X -0.007,Y -580.895,Z 1070.437,A 0.000,B 0.000,C 90.000,E1 294.695} C_DIS
LIN {X -0.073,Y -579.687,Z 1070.437,A 0.000,B 0.000,C 90.000,E1 294.567} C_DIS
LIN {X 0.203,Y -573.092,Z 1070.433,A 0.000,B 0.000,C 90.000,E1 293.898} C_DIS
LIN {X 0.199,Y -571.549,Z 1070.432,A 0.000,B 0.000,C 90.000,E1 293.770} C_DIS
LIN {X 0.196,Y -569.763,Z 1070.432,A 0.000,B 0.000,C 90.000,E1 293.643} C_DIS
LIN {X 0.200,Y -564.711,Z 1070.430,A 0.000,B 0.000,C 90.000,E1 293.334} C_DIS
LIN {X -0.125,Y -561.302,Z 1070.429,A 0.000,B 0.000,C 90.000,E1 293.206} C_DIS
LIN {X -0.053,Y -557.324,Z 1070.428,A 0.000,B 0.000,C 90.000,E1 293.131} C_DIS
LIN {X 0.239,Y -554.210,Z 1070.428,A 0.000,B 0.000,C 90.000,E1 293.078} C_DIS
LIN {X -0.017,Y -550.495,Z 1070.427,A 0.000,B 0.000,C 90.000,E1 292.950} C_DIS
LIN {X -0.136,Y -549.006,Z 1070.427,A 0.000,B 0.000,C 90.000,E1 292.898} C_DIS
LIN {X -0.135,Y -548.237,Z 1070.427,A 0.000,B 0.000,C 90.000,E1 292.823} C_DIS
LIN {X -0.288,Y -546.478,Z 1070.425,A 0.000,B 0.000,C 90.000,E1 292.589} C_DIS
LIN {X 0.095,Y -545.923,Z 1070.425,A 0.000,B 0.000,C 90.000,E1 292.408} C_DIS
LIN {X -0.076,Y -544.451,Z 1070.422,A 0.000,B 0.000,C 90.000,E1 291.950} C_DIS
LIN {X -0.250,Y -543.995,Z 1070.420,A 0.000,B 0.000,C 90.000,E1 291.589} C_DIS
LIN {X -0.007,Y -543.926,Z 1070.418,A 0.000,B 0.000,C 90.000,E1 291.280} C_DIS
LIN {X 0.236,Y -543.645,Z 1070.417,A 0.000,B 0.000,C 90.000,E1 290.972} C_DIS
LIN {X -0.091,Y -543.384,Z 1070.416,A 0.000,B 0.000,C 90.000,E1 290.865} C_DIS
LIN {X -0.013,Y -543.107,Z 1070.410,A 0.000,B 0.000,C 90.000,E1 289.866} C_DIS
LIN {X -0.155,Y -543.180,Z 1070.401,A 0.000,B 0.000,C 90.000,E1 288.181} C_DIS
LIN {X 0.160,Y -543.273,Z 1070.393,A 0.000,B 0.000,C 90.000,E1 286.732} C_DIS
LIN {X 0.167,Y -543.002,Z 1070.385,A 0.000,B 0.000,C 90.000,E1 285.315} C_DIS
LIN {X -0.212,Y -542.524,Z 1070.377,A 0.000,B 0.000,C 90.000,E1 283.939} C_DIS
LIN {X 0.108,Y -542.152,Z 1070.371,A 0.000,B 0.000,C 90.000,E1 282.771} C_DIS
LIN {X 0.064,Y -541.245,Z 1070.362,A 0.000,B 0.000,C 90.000,E1 281.074} C_DIS
LIN {X -0.084,Y -540.432,Z 1070.354,A 0.000,B 0.000,C 90.000,E1 279.670} C_DIS
LIN {X 0.189,Y -539.689,Z 1070.346,A 0.000,B 0.000,C 90.000,E1 278.219} C_DIS
LIN {X -0.050,Y -538.392,Z 1070.333,A 0.000,B 0.000,C 90.000,E1 275.967} C_DIS
LIN {X 0.100,Y -537.330,Z 1070.322,A 0.000,B 0.000,C 90.000,E1 273.955} C_DIS
LIN {X 0.163,Y -536.293,Z 1070.311,A 0.000,B 0.000,C 90.000,E1 271.949} C_DIS
LIN {X 0.202,Y -535.469,Z 1070.303,A 0.000,B 0.000,C 90.000,E1 270.516} C_DIS
LIN {X 0.213,Y -534.684,Z 1070.295,A 0.000,B 0.000,C 90.000,E1 269.083} C_DIS
LIN {X 0.217,Y -533.675,Z 1070.286,A 0.000,B 0.000,C 90.000,E1 267.364} C_DIS
LIN {X 0.200,Y -532.799,Z 1070.278,A 0.000,B 0.000,C 90.000,E1 265.931} C_DIS
LIN {X 0.250,Y -531.784,Z 1070.270,A 0.000,B 0.000,C 90.000,E1 264.489} C_DIS
LIN {X 0.230,Y -530.526,Z 1070.262,A 0.000,B 0.000,C 90.000,E1 263.053} C_DIS
LIN {X -0.241,Y -529.346,Z 1070.255,A 0.000,B 0.000,C 90.000,E1 261.951} C_DIS
LIN {X -0.170,Y -527.806,Z 1070.247,A 0.000,B 0.000,C 90.000,E1 260.500} C_DIS
LIN {X -0.109,Y -525.900,Z 1070.238,A 0.000,B 0.000,C 90.000,E1 258.757} C_DIS
LIN {X 0.114,Y -524.083,Z 1070.228,A 0.000,B 0.000,C 90.000,E1 256.992} C_DIS
LIN {X -0.206,Y -522.279,Z 1070.218,A 0.000,B 0.000,C 90.000,E1 255.283} C_DIS
LIN {X -0.067,Y -521.140,Z 1070.212,A 0.000,B 0.000,C 90.000,E1 254.102} C_DIS
LIN {X -0.180,Y -519.292,Z 1070.202,A 0.000,B 0.000,C 90.000,E1 252.362} C_DIS
LIN {X 0.214,Y -518.064,Z 1070.195,A 0.000,B 0.000,C 90.000,E1 251.148} C_DIS
LIN {X -0.153,Y -515.710,Z 1070.184,A 0.000,B 0.000,C 90.000,E1 249.135} C_DIS
LIN {X -0.171,Y -513.705,Z 1070.176,A 0.000,B 0.000,C 90.000,E1 247.667} C_DIS
LIN {X -0.041,Y -511.638,Z 1070.168,A 0.000,B 0.000,C 90.000,E1 246.177} C_DIS
LIN {X -0.209,Y -509.406,Z 1070.159,A 0.000,B 0.000,C 90.000,E1 244.717} C_DIS
LIN {X 0.040,Y -507.020,Z 1070.151,A 0.000,B 0.000,C 90.000,E1 243.204} C_DIS
LIN {X -0.123,Y -504.021,Z 1070.141,A 0.000,B 0.000,C 90.000,E1 241.435} C_DIS
LIN {X 0.176,Y -501.983,Z 1070.135,A 0.000,B 0.000,C 90.000,E1 240.205} C_DIS
LIN {X -0.139,Y -499.294,Z 1070.126,A 0.000,B 0.000,C 90.000,E1 238.742} C_DIS
LIN {X -0.240,Y -496.541,Z 1070.118,A 0.000,B 0.000,C 90.000,E1 237.248} C_DIS
LIN {X 0.027,Y -494.206,Z 1070.111,A 0.000,B 0.000,C 90.000,E1 236.008} C_DIS
LIN {X 0.104,Y -491.276,Z 1070.103,A 0.000,B 0.000,C 90.000,E1 234.482} C_DIS
LIN {X -0.147,Y -487.420,Z 1070.093,A 0.000,B 0.000,C 90.000,E1 232.683} C_DIS
LIN {X 0.069,Y -483.965,Z 1070.084,A 0.000,B 0.000,C 90.000,E1 231.126} C_DIS
LIN {X -0.047,Y -481.272,Z 1070.077,A 0.000,B 0.000,C 90.000,E1 229.908} C_DIS
LIN {X 0.183,Y -476.647,Z 1070.065,A 0.000,B 0.000,C 90.000,E1 227.715} C_DIS
LIN {X -0.089,Y -472.377,Z 1070.053,A 0.000,B 0.000,C 90.000,E1 225.567} C_DIS
LIN {X -0.064,Y -467.737,Z 1070.039,A 0.000,B 0.000,C 90.000,E1 223.056} C_DIS
LIN {X -0.003,Y -464.704,Z 1070.030,A 0.000,B 0.000,C 90.000,E1 221.472} C_DIS
LIN {X 0.050,Y -460.801,Z 1070.020,A 0.000,B 0.000,C 90.000,E1 219.564} C_DIS
LIN {X 0.048,Y -457.658,Z 1070.011,A 0.000,B 0.000,C 90.000,E1 217.971} C_DIS
LIN {X -0.011,Y -454.473,Z 1070.002,A 0.000,B 0.000,C 90.000,E1 216.377} C_DIS
LIN {X -0.064,Y -450.423,Z 1069.991,A 0.000,B 0.000,C 90.000,E1 214.452} C_DIS
LIN {X -0.211,Y -445.246,Z 1069.977,A 0.000,B 0.000,C 90.000,E1 211.878} C_DIS
LIN {X 0.096,Y -442.140,Z 1069.968,A 0.000,B 0.000,C 90.000,E1 210.207} C_DIS
LIN {X 0.075,Y -439.548,Z 1069.961,A 0.000,B 0.000,C 90.000,E1 208.899} C_DIS
LIN {X 0.119,Y -434.002,Z 1069.944,A 0.000,B 0.000,C 90.000,E1 205.924} C_DIS
LIN {X 0.159,Y -429.429,Z 1069.929,A 0.000,B 0.000,C 90.000,E1 203.259} C_DIS
LIN {X 0.133,Y -425.079,Z 1069.913,A 0.000,B 0.000,C 90.000,E1 200.248} C_DIS
LIN {X 0.100,Y -423.937,Z 1069.905,A 0.000,B 0.000,C 90.000,E1 198.906} C_DIS
LIN {X 0.259,Y -423.482,Z 1069.900,A 0.000,B 0.000,C 90.000,E1 197.873} C_DIS
LIN {X 0.098,Y -423.625,Z 1069.896,A 0.000,B 0.000,C 90.000,E1 197.221} C_DIS
LIN {X 0.062,Y -424.123,Z 1069.892,A 0.000,B 0.000,C 90.000,E1 196.551} C_DIS
LIN {X -0.094,Y -425.087,Z 1069.888,A 0.000,B 0.000,C 90.000,E1 195.898} C_DIS
LIN {X 0.168,Y -426.628,Z 1069.885,A 0.000,B 0.000,C 90.000,E1 195.190} C_DIS
LIN {X 0.031,Y -428.578,Z 1069.881,A 0.000,B 0.000,C 90.000,E1 194.537} C_DIS
LIN {X -0.193,Y -430.365,Z 1069.878,A 0.000,B 0.000,C 90.000,E1 194.064} C_DIS
LIN {X 0.223,Y -433.848,Z 1069.873,A 0.000,B 0.000,C 90.000,E1 193.175} C_DIS
LIN {X 0.179,Y -438.541,Z 1069.868,A 0.000,B 0.000,C 90.000,E1 192.187} C_DIS
LIN {X -0.120,Y -448.329,Z 1069.858,A 0.000,B 0.000,C 90.000,E1 190.423} C_DIS
LIN {X 0.005,Y -462.485,Z 1069.844,A 0.000,B 0.000,C 90.000,E1 187.992} C_DIS
LIN {X -0.138,Y -471.900,Z 1069.836,A 0.000,B 0.000,C 90.000,E1 186.429} C_DIS
LIN {X -0.134,Y -478.101,Z 1069.830,A 0.000,B 0.000,C 90.000,E1 185.334} C_DIS
LIN {X -0.088,Y -484.156,Z 1069.824,A 0.000,B 0.000,C 90.000,E1 184.245} C_DIS
LIN {X 0.051,Y -490.170,Z 1069.818,A 0.000,B 0.000,C 90.000,E1 183.154} C_DIS
LIN {X -0.225,Y -495.972,Z 1069.812,A 0.000,B 0.000,C 90.000,E1 182.121} C_DIS
LIN {X -0.121,Y -500.855,Z 1069.807,A 0.000,B 0.000,C 90.000,E1 181.203} C_DIS
LIN {X -0.079,Y -507.271,Z 1069.800,A 0.000,B 0.000,C 90.000,E1 180.000} C_DIS
LIN {X 0.201,Y -516.008,Z 1069.791,A 0.000,B 0.000,C 90.000,E1 178.339} C_DIS
LIN {X 0.253,Y -521.453,Z 1069.785,A 0.000,B 0.000,C 90.000,E1 177.306} C_DIS
LIN {X 0.100,Y -529.106,Z 1069.777,A 0.000,B 0.000,C 90.000,E1 175.869} C_DIS
LIN {X 0.091,Y -536.690,Z 1069.769,A 0.000,B 0.000,C 90.000,E1 174.432} C_DIS
LIN {X 0.010,Y -544.936,Z 1069.760,A 0.000,B 0.000,C 90.000,E1 172.875} C_DIS
LIN {X 0.231,Y -550.829,Z 1069.754,A 0.000,B 0.000,C 90.000,E1 171.724} C_DIS
LIN {X -0.101,Y -557.290,Z 1069.747,A 0.000,B 0.000,C 90.000,E1 170.500} C_DIS
LIN {X -0.021,Y -564.236,Z 1069.740,A 0.000,B 0.000,C 90.000,E1 169.106} C_DIS
LIN {X 0.236,Y -568.982,Z 1069.734,A 0.000,B 0.000,C 90.000,E1 168.117} C_DIS
LIN {X -0.080,Y -572.275,Z 1069.730,A 0.000,B 0.000,C 90.000,E1 167.465} C_DIS
LIN {X 0.264,Y -579.183,Z 1069.722,A 0.000,B 0.000,C 90.000,E1 165.936} C_DIS
LIN {X 0.268,Y -583.389,Z 1069.717,A 0.000,B 0.000,C 90.000,E1 164.991} C_DIS
LIN {X -0.009,Y -586.870,Z 1069.712,A 0.000,B 0.000,C 90.000,E1 164.212} C_DIS
LIN {X 0.003,Y -591.317,Z 1069.706,A 0.000,B 0.000,C 90.000,E1 163.142} C_DIS
LIN {X 0.249,Y -595.448,Z 1069.700,A 0.000,B 0.000,C 90.000,E1 162.054} C_DIS
LIN {X -0.203,Y -599.399,Z 1069.695,A 0.000,B 0.000,C 90.000,E1 161.040} C_DIS
LIN {X 0.066,Y -603.964,Z 1069.687,A 0.000,B 0.000,C 90.000,E1 159.699} C_DIS
LIN {X -0.151,Y -608.179,Z 1069.680,A 0.000,B 0.000,C 90.000,E1 158.411} C_DIS
LIN {X -0.027,Y -611.404,Z 1069.674,A 0.000,B 0.000,C 90.000,E1 157.358} C_DIS
LIN {X 0.110,Y -615.163,Z 1069.667,A 0.000,B 0.000,C 90.000,E1 156.049} C_DIS
LIN {X -0.257,Y -618.694,Z 1069.660,A 0.000,B 0.000,C 90.000,E1 154.793} C_DIS
LIN {X -0.291,Y -620.680,Z 1069.656,A 0.000,B 0.000,C 90.000,E1 154.024} C_DIS
LIN {X -0.288,Y -625.187,Z 1069.646,A 0.000,B 0.000,C 90.000,E1 152.231} C_DIS
LIN {X 0.086,Y -628.832,Z 1069.637,A 0.000,B 0.000,C 90.000,E1 150.667} C_DIS
LIN {X -0.042,Y -631.750,Z 1069.630,A 0.000,B 0.000,C 90.000,E1 149.410} C_DIS
LIN {X 0.235,Y -635.070,Z 1069.622,A 0.000,B 0.000,C 90.000,E1 147.867} C_DIS
LIN {X 0.006,Y -637.736,Z 1069.615,A 0.000,B 0.000,C 90.000,E1 146.628} C_DIS
LIN {X 0.220,Y -640.871,Z 1069.606,A 0.000,B 0.000,C 90.000,E1 145.102} C_DIS
LIN {X -0.028,Y -643.886,Z 1069.598,A 0.000,B 0.000,C 90.000,E1 143.623} C_DIS
LIN {X 0.166,Y -646.962,Z 1069.590,A 0.000,B 0.000,C 90.000,E1 142.110} C_DIS
LIN {X -0.089,Y -649.921,Z 1069.581,A 0.000,B 0.000,C 90.000,E1 140.642} C_DIS
LIN {X 0.129,Y -653.005,Z 1069.573,A 0.000,B 0.000,C 90.000,E1 139.138} C_DIS
LIN {X 0.366,Y -656.669,Z 1069.563,A 0.000,B 0.000,C 90.000,E1 137.391} C_DIS
LIN {X -0.288,Y -660.500,Z 1069.554,A 0.000,B 0.000,C 90.000,E1 135.729} C_DIS
LIN {X -0.395,Y -664.655,Z 1069.544,A 0.000,B 0.000,C 90.000,E1 134.028} C_DIS
LIN {X 0.067,Y -669.134,Z 1069.535,A 0.000,B 0.000,C 90.000,E1 132.285} C_DIS
LIN {X 0.162,Y -672.842,Z 1069.527,A 0.000,B 0.000,C 90.000,E1 130.825} C_DIS
LIN {X -0.129,Y -676.093,Z 1069.520,A 0.000,B 0.000,C 90.000,E1 129.644} C_DIS
LIN {X -0.189,Y -680.930,Z 1069.510,A 0.000,B 0.000,C 90.000,E1 127.729} C_DIS
LIN {X 0.185,Y -684.070,Z 1069.503,A 0.000,B 0.000,C 90.000,E1 126.503} C_DIS
LIN {X 0.001,Y -685.955,Z 1069.499,A 0.000,B 0.000,C 90.000,E1 125.804} C_DIS
LIN {X -0.315,Y -689.397,Z 1069.491,A 0.000,B 0.000,C 90.000,E1 124.405} C_DIS
LIN {X 0.147,Y -691.700,Z 1069.486,A 0.000,B 0.000,C 90.000,E1 123.420} C_DIS
LIN {X -0.101,Y -694.572,Z 1069.479,A 0.000,B 0.000,C 90.000,E1 122.260} C_DIS
LIN {X -0.076,Y -697.226,Z 1069.473,A 0.000,B 0.000,C 90.000,E1 121.082} C_DIS
LIN {X 0.100,Y -699.315,Z 1069.468,A 0.000,B 0.000,C 90.000,E1 120.129} C_DIS
LIN {X 0.285,Y -700.513,Z 1069.464,A 0.000,B 0.000,C 90.000,E1 119.411} C_DIS
LIN {X -0.130,Y -701.417,Z 1069.460,A 0.000,B 0.000,C 90.000,E1 118.743} C_DIS
LIN {X -0.170,Y -703.601,Z 1069.447,A 0.000,B 0.000,C 90.000,E1 116.411} C_DIS
LIN {X -0.261,Y -704.306,Z 1069.443,A 0.000,B 0.000,C 90.000,E1 115.720} C_DIS
LIN {X -0.340,Y -704.750,Z 1069.439,A 0.000,B 0.000,C 90.000,E1 115.027} C_DIS
LIN {X -0.054,Y -704.865,Z 1069.438,A 0.000,B 0.000,C 90.000,E1 114.771} C_DIS
LIN {X 0.232,Y -704.811,Z 1069.436,A 0.000,B 0.000,C 90.000,E1 114.515} C_DIS
LIN {X -0.129,Y -704.411,Z 1069.434,A 0.000,B 0.000,C 90.000,E1 114.079} C_DIS
LIN {X 0.155,Y -703.808,Z 1069.432,A 0.000,B 0.000,C 90.000,E1 113.823} C_DIS
LIN {X -0.208,Y -702.284,Z 1069.430,A 0.000,B 0.000,C 90.000,E1 113.387} C_DIS
LIN {X -0.070,Y -701.589,Z 1069.429,A 0.000,B 0.000,C 90.000,E1 113.259} C_DIS
LIN {X 0.195,Y -698.083,Z 1069.427,A 0.000,B 0.000,C 90.000,E1 112.770} C_DIS
LIN {X 0.326,Y -696.911,Z 1069.426,A 0.000,B 0.000,C 90.000,E1 112.642} C_DIS
LIN {X -0.187,Y -695.098,Z 1069.425,A 0.000,B 0.000,C 90.000,E1 112.567} C_DIS
LIN {X 0.098,Y -687.696,Z 1069.423,A 0.000,B 0.000,C 90.000,E1 112.206} C_DIS
LIN {X -0.149,Y -685.621,Z 1069.423,A 0.000,B 0.000,C 90.000,E1 112.153} C_DIS
LIN {X 0.095,Y -682.628,Z 1069.423,A 0.000,B 0.000,C 90.000,E1 112.078} C_DIS
LIN {X -0.239,Y -676.064,Z 1069.422,A 0.000,B 0.000,C 90.000,E1 112.025} C_DIS
LIN {X -0.262,Y -607.719,Z 1069.422,A 0.000,B 0.000,C 90.000,E1 112.025} C_DIS
LIN {X 0.055,Y -603.913,Z 1069.421,A 0.000,B 0.000,C 90.000,E1 111.844} C_DIS
LIN {X 0.075,Y -602.250,Z 1069.421,A 0.000,B 0.000,C 90.000,E1 111.770} C_DIS
LIN {X 0.261,Y -596.367,Z 1069.419,A 0.000,B 0.000,C 90.000,E1 111.408} C_DIS
LIN {X -0.077,Y -589.538,Z 1069.416,A 0.000,B 0.000,C 90.000,E1 110.918} C_DIS
LIN {X -0.096,Y -579.991,Z 1069.412,A 0.000,B 0.000,C 90.000,E1 110.120} C_DIS
LIN {X 0.252,Y -574.363,Z 1069.409,A 0.000,B 0.000,C 90.000,E1 109.631} C_DIS
LIN {X 0.066,Y -568.471,Z 1069.407,A 0.000,B 0.000,C 90.000,E1 109.214} C_DIS
LIN {X 0.017,Y -560.250,Z 1069.404,A 0.000,B 0.000,C 90.000,E1 108.725} C_DIS
LIN {X -0.018,Y -553.874,Z 1069.402,A 0.000,B 0.000,C 90.000,E1 108.362} C_DIS
LIN {X 0.120,Y -549.578,Z 1069.400,A 0.000,B 0.000,C 90.000,E1 108.055} C_DIS
LIN {X -0.224,Y -547.673,Z 1069.399,A 0.000,B 0.000,C 90.000,E1 107.873} C_DIS
LIN {X 0.256,Y -547.660,Z 1069.399,A 0.000,B 0.000,C 90.000,E1 107.819} C_DIS
LIN {X 0.215,Y -547.309,Z 1069.397,A 0.000,B 0.000,C 90.000,E1 107.511} C_DIS
LIN {X 0.062,Y -548.666,Z 1069.384,A 0.000,B 0.000,C 90.000,E1 105.134} C_DIS
LIN {X -0.007,Y -550.122,Z 1069.373,A 0.000,B 0.000,C 90.000,E1 103.175} C_DIS
LIN {X 0.240,Y -551.815,Z 1069.362,A 0.000,B 0.000,C 90.000,E1 101.186} C_DIS
LIN {X 0.132,Y -554.465,Z 1069.348,A 0.000,B 0.000,C 90.000,E1 98.681} C_DIS
LIN {X 0.169,Y -556.367,Z 1069.339,A 0.000,B 0.000,C 90.000,E1 97.004} C_DIS
LIN {X -0.013,Y -557.658,Z 1069.333,A 0.000,B 0.000,C 90.000,E1 95.910} C_DIS
LIN {X -0.101,Y -558.983,Z 1069.325,A 0.000,B 0.000,C 90.000,E1 94.531} C_DIS
LIN {X -0.170,Y -559.850,Z 1069.318,A 0.000,B 0.000,C 90.000,E1 93.151} C_DIS
LIN {X -0.260,Y -560.589,Z 1069.310,A 0.000,B 0.000,C 90.000,E1 91.776} C_DIS
LIN {X 0.213,Y -561.194,Z 1069.302,A 0.000,B 0.000,C 90.000,E1 90.344} C_DIS
LIN {X 0.239,Y -561.834,Z 1069.293,A 0.000,B 0.000,C 90.000,E1 88.682} C_DIS
LIN {X -0.051,Y -562.694,Z 1069.281,A 0.000,B 0.000,C 90.000,E1 86.502} C_DIS
LIN {X -0.047,Y -563.190,Z 1069.273,A 0.000,B 0.000,C 90.000,E1 85.122} C_DIS
LIN {X -0.035,Y -563.625,Z 1069.265,A 0.000,B 0.000,C 90.000,E1 83.742} C_DIS
LIN {X 0.201,Y -564.049,Z 1069.256,A 0.000,B 0.000,C 90.000,E1 82.064} C_DIS
LIN {X 0.220,Y -564.836,Z 1069.244,A 0.000,B 0.000,C 90.000,E1 79.859} C_DIS
LIN {X -0.034,Y -565.927,Z 1069.230,A 0.000,B 0.000,C 90.000,E1 77.409} C_DIS
LIN {X 0.019,Y -566.887,Z 1069.221,A 0.000,B 0.000,C 90.000,E1 75.755} C_DIS
LIN {X 0.160,Y -569.042,Z 1069.204,A 0.000,B 0.000,C 90.000,E1 72.725} C_DIS
LIN {X 0.020,Y -570.777,Z 1069.192,A 0.000,B 0.000,C 90.000,E1 70.550} C_DIS
LIN {X -0.219,Y -571.924,Z 1069.184,A 0.000,B 0.000,C 90.000,E1 69.209} C_DIS
LIN {X -0.231,Y -573.027,Z 1069.177,A 0.000,B 0.000,C 90.000,E1 67.847} C_DIS
LIN {X -0.224,Y -574.069,Z 1069.169,A 0.000,B 0.000,C 90.000,E1 66.485} C_DIS
LIN {X -0.179,Y -574.744,Z 1069.165,A 0.000,B 0.000,C 90.000,E1 65.665} C_DIS
LIN {X -0.068,Y -575.729,Z 1069.156,A 0.000,B 0.000,C 90.000,E1 64.024} C_DIS
LIN {X -0.199,Y -576.675,Z 1069.147,A 0.000,B 0.000,C 90.000,E1 62.410} C_DIS
LIN {X -0.314,Y -577.579,Z 1069.138,A 0.000,B 0.000,C 90.000,E1 60.795} C_DIS
LIN {X 0.011,Y -578.219,Z 1069.130,A 0.000,B 0.000,C 90.000,E1 59.410} C_DIS
LIN {X -0.153,Y -578.790,Z 1069.123,A 0.000,B 0.000,C 90.000,E1 58.074} C_DIS
LIN {X -0.001,Y -579.395,Z 1069.115,A 0.000,B 0.000,C 90.000,E1 56.707} C_DIS
LIN {X -0.152,Y -580.021,Z 1069.106,A 0.000,B 0.000,C 90.000,E1 55.102} C_DIS
LIN {X 0.181,Y -580.379,Z 1069.100,A 0.000,B 0.000,C 90.000,E1 53.989} C_DIS
LIN {X 0.215,Y -580.561,Z 1069.093,A 0.000,B 0.000,C 90.000,E1 52.637} C_DIS
LIN {X -0.020,Y -580.577,Z 1069.087,A 0.000,B 0.000,C 90.000,E1 51.582} C_DIS
LIN {X -0.329,Y -580.472,Z 1069.082,A 0.000,B 0.000,C 90.000,E1 50.803} C_DIS
LIN {X 0.308,Y -579.741,Z 1069.072,A 0.000,B 0.000,C 90.000,E1 48.852} C_DIS
LIN {X -0.210,Y -579.100,Z 1069.064,A 0.000,B 0.000,C 90.000,E1 47.553} C_DIS
LIN {X -0.072,Y -578.429,Z 1069.058,A 0.000,B 0.000,C 90.000,E1 46.458} C_DIS
LIN {X 0.051,Y -577.597,Z 1069.052,A 0.000,B 0.000,C 90.000,E1 45.364} C_DIS
LIN {X 0.027,Y -576.789,Z 1069.048,A 0.000,B 0.000,C 90.000,E1 44.555} C_DIS
LIN {X 0.125,Y -575.393,Z 1069.042,A 0.000,B 0.000,C 90.000,E1 43.461} C_DIS
LIN {X 0.207,Y -573.859,Z 1069.036,A 0.000,B 0.000,C 90.000,E1 42.366} C_DIS
LIN {X -0.114,Y -572.201,Z 1069.030,A 0.000,B 0.000,C 90.000,E1 41.310} C_DIS
LIN {X 0.093,Y -571.216,Z 1069.026,A 0.000,B 0.000,C 90.000,E1 40.744} C_DIS
LIN {X 0.169,Y -568.849,Z 1069.020,A 0.000,B 0.000,C 90.000,E1 39.644} C_DIS
LIN {X 0.219,Y -566.206,Z 1069.014,A 0.000,B 0.000,C 90.000,E1 38.543} C_DIS
LIN {X 0.008,Y -564.749,Z 1069.011,A 0.000,B 0.000,C 90.000,E1 38.016} C_DIS
LIN {X 0.337,Y -562.289,Z 1069.007,A 0.000,B 0.000,C 90.000,E1 37.156} C_DIS
LIN {X -0.243,Y -560.476,Z 1069.004,A 0.000,B 0.000,C 90.000,E1 36.664} C_DIS
LIN {X -0.049,Y -558.442,Z 1069.000,A 0.000,B 0.000,C 90.000,E1 36.091} C_DIS
LIN {X -0.033,Y -553.981,Z 1068.994,A 0.000,B 0.000,C 90.000,E1 34.978} C_DIS
LIN {X 0.171,Y -550.242,Z 1068.990,A 0.000,B 0.000,C 90.000,E1 34.119} C_DIS
LIN {X 0.016,Y -546.167,Z 1068.985,A 0.000,B 0.000,C 90.000,E1 33.293} C_DIS
LIN {X -0.210,Y -543.242,Z 1068.982,A 0.000,B 0.000,C 90.000,E1 32.752} C_DIS
LIN {X -0.118,Y -537.943,Z 1068.976,A 0.000,B 0.000,C 90.000,E1 31.750} C_DIS
LIN {X -0.117,Y -534.697,Z 1068.973,A 0.000,B 0.000,C 90.000,E1 31.180} C_DIS
LIN {X 0.036,Y -531.220,Z 1068.970,A 0.000,B 0.000,C 90.000,E1 30.590} C_DIS
LIN {X 0.014,Y -526.529,Z 1068.966,A 0.000,B 0.000,C 90.000,E1 29.873} C_DIS
LIN {X -0.188,Y -523.532,Z 1068.964,A 0.000,B 0.000,C 90.000,E1 29.461} C_DIS
LIN {X 0.179,Y -518.168,Z 1068.960,A 0.000,B 0.000,C 90.000,E1 28.693} C_DIS
LIN {X -0.073,Y -514.781,Z 1068.957,A 0.000,B 0.000,C 90.000,E1 28.281} C_DIS
LIN {X -0.067,Y -509.874,Z 1068.954,A 0.000,B 0.000,C 90.000,E1 27.692} C_DIS
LIN {X -0.228,Y -504.852,Z 1068.951,A 0.000,B 0.000,C 90.000,E1 27.129} C_DIS
LIN {X -0.061,Y -500.868,Z 1068.948,A 0.000,B 0.000,C 90.000,E1 26.668} C_DIS
LIN {X 0.099,Y -491.378,Z 1068.943,A 0.000,B 0.000,C 90.000,E1 25.668} C_DIS
LIN {X -0.092,Y -486.050,Z 1068.940,A 0.000,B 0.000,C 90.000,E1 25.155} C_DIS
LIN {X -0.118,Y -477.481,Z 1068.935,A 0.000,B 0.000,C 90.000,E1 24.335} C_DIS
LIN {X -0.014,Y -468.663,Z 1068.931,A 0.000,B 0.000,C 90.000,E1 23.515} C_DIS
LIN {X 0.028,Y -459.518,Z 1068.926,A 0.000,B 0.000,C 90.000,E1 22.717} C_DIS
LIN {X 0.008,Y -444.367,Z 1068.919,A 0.000,B 0.000,C 90.000,E1 21.408} C_DIS
LIN {X -0.151,Y -428.347,Z 1068.911,A 0.000,B 0.000,C 90.000,E1 19.939} C_DIS
LIN {X 0.183,Y -414.156,Z 1068.902,A 0.000,B 0.000,C 90.000,E1 18.417} C_DIS
LIN {X -0.133,Y -402.172,Z 1068.895,A 0.000,B 0.000,C 90.000,E1 17.040} C_DIS
LIN {X 0.152,Y -397.801,Z 1068.891,A 0.000,B 0.000,C 90.000,E1 16.386} C_DIS
LIN {X -0.033,Y -393.702,Z 1068.887,A 0.000,B 0.000,C 90.000,E1 15.662} C_DIS
LIN {X 0.064,Y -392.707,Z 1068.885,A 0.000,B 0.000,C 90.000,E1 15.315} C_DIS
LIN {X -0.004,Y -392.269,Z 1068.883,A 0.000,B 0.000,C 90.000,E1 15.009} C_DIS
LIN {X -0.057,Y -391.906,Z 1068.881,A 0.000,B 0.000,C 90.000,E1 14.662} C_DIS
LIN {X -0.011,Y -391.889,Z 1068.880,A 0.000,B 0.000,C 90.000,E1 14.300} C_DIS
LIN {X 0.030,Y -391.993,Z 1068.878,A 0.000,B 0.000,C 90.000,E1 13.939} C_DIS
LIN {X -0.040,Y -394.029,Z 1068.868,A 0.000,B 0.000,C 90.000,E1 12.175} C_DIS
LIN {X 0.098,Y -400.413,Z 1068.846,A 0.000,B 0.000,C 90.000,E1 8.276} C_DIS
LIN {X -0.060,Y -405.559,Z 1068.833,A 0.000,B 0.000,C 90.000,E1 5.853} C_DIS
LIN {X -0.132,Y -409.044,Z 1068.824,A 0.000,B 0.000,C 90.000,E1 4.302} C_DIS
LIN {X -0.118,Y -410.386,Z 1068.822,A 0.000,B 0.000,C 90.000,E1 3.898} C_DIS
LIN {X -0.132,Y -411.709,Z 1068.820,A 0.000,B 0.000,C 90.000,E1 3.555} C_DIS
LIN {X 0.168,Y -417.102,Z 1068.815,A 0.000,B 0.000,C 90.000,E1 2.751} C_DIS
LIN {X 0.056,Y -420.693,Z 1068.814,A 0.000,B 0.000,C 90.000,E1 2.465} C_DIS
LIN {X 0.174,Y -428.967,Z 1068.811,A 0.000,B 0.000,C 90.000,E1 1.892} C_DIS
LIN {X 0.123,Y -440.490,Z 1068.807,A 0.000,B 0.000,C 90.000,E1 1.146} C_DIS
LIN {X 0.175,Y -462.187,Z 1068.799,A 0.000,B 0.000,C 90.000,E1 359.771} C_DIS
LIN {X -0.045,Y -478.444,Z 1068.793,A 0.000,B 0.000,C 90.000,E1 358.797} C_DIS
LIN {X -0.124,Y -489.675,Z 1068.789,A 0.000,B 0.000,C 90.000,E1 358.108} C_DIS
LIN {X -0.175,Y -497.577,Z 1068.787,A 0.000,B 0.000,C 90.000,E1 357.593} C_DIS
LIN {X 0.132,Y -505.444,Z 1068.784,A 0.000,B 0.000,C 90.000,E1 357.020} C_DIS
LIN {X -0.210,Y -511.514,Z 1068.781,A 0.000,B 0.000,C 90.000,E1 356.617} C_DIS
LIN {X -0.107,Y -517.332,Z 1068.779,A 0.000,B 0.000,C 90.000,E1 356.159} C_DIS
LIN {X -0.237,Y -523.152,Z 1068.776,A 0.000,B 0.000,C 90.000,E1 355.698} C_DIS
LIN {X 0.268,Y -530.103,Z 1068.772,A 0.000,B 0.000,C 90.000,E1 355.008} C_DIS
LIN {X 0.053,Y -536.730,Z 1068.769,A 0.000,B 0.000,C 90.000,E1 354.375} C_DIS
LIN {X 0.024,Y -543.033,Z 1068.765,A 0.000,B 0.000,C 90.000,E1 353.685} C_DIS
LIN {X 0.111,Y -547.837,Z 1068.762,A 0.000,B 0.000,C 90.000,E1 353.109} C_DIS
LIN {X 0.050,Y -552.996,Z 1068.758,A 0.000,B 0.000,C 90.000,E1 352.413} C_DIS
LIN {X -0.044,Y -557.640,Z 1068.754,A 0.000,B 0.000,C 90.000,E1 351.724} C_DIS
LIN {X 0.229,Y -561.018,Z 1068.751,A 0.000,B 0.000,C 90.000,E1 351.141} C_DIS
LIN {X 0.290,Y -564.823,Z 1068.747,A 0.000,B 0.000,C 90.000,E1 350.443} C_DIS
LIN {X -0.176,Y -568.301,Z 1068.743,A 0.000,B 0.000,C 90.000,E1 349.803} C_DIS
LIN {X 0.188,Y -570.875,Z 1068.740,A 0.000,B 0.000,C 90.000,E1 349.218} C_DIS
LIN {X -0.268,Y -575.708,Z 1068.734,A 0.000,B 0.000,C 90.000,E1 348.173} C_DIS
LIN {X -0.208,Y -579.050,Z 1068.730,A 0.000,B 0.000,C 90.000,E1 347.353} C_DIS
LIN {X 0.250,Y -583.258,Z 1068.724,A 0.000,B 0.000,C 90.000,E1 346.228} C_DIS
LIN {X -0.178,Y -586.233,Z 1068.719,A 0.000,B 0.000,C 90.000,E1 345.463} C_DIS
LIN {X 0.074,Y -590.965,Z 1068.712,A 0.000,B 0.000,C 90.000,E1 344.102} C_DIS
LIN {X 0.004,Y -595.483,Z 1068.704,A 0.000,B 0.000,C 90.000,E1 342.779} C_DIS
LIN {X 0.122,Y -598.870,Z 1068.698,A 0.000,B 0.000,C 90.000,E1 341.710} C_DIS
LIN {X -0.099,Y -601.963,Z 1068.693,A 0.000,B 0.000,C 90.000,E1 340.678} C_DIS
LIN {X 0.210,Y -605.538,Z 1068.685,A 0.000,B 0.000,C 90.000,E1 339.337} C_DIS
LIN {X 0.012,Y -608.757,Z 1068.678,A 0.000,B 0.000,C 90.000,E1 338.050} C_DIS
LIN {X 0.139,Y -611.014,Z 1068.672,A 0.000,B 0.000,C 90.000,E1 336.997} C_DIS
LIN {X -0.018,Y -613.027,Z 1068.667,A 0.000,B 0.000,C 90.000,E1 335.973} C_DIS
LIN {X 0.165,Y -614.748,Z 1068.661,A 0.000,B 0.000,C 90.000,E1 334.921} C_DIS
LIN {X 0.051,Y -616.573,Z 1068.654,A 0.000,B 0.000,C 90.000,E1 333.640} C_DIS
LIN {X 0.000,Y -617.570,Z 1068.649,A 0.000,B 0.000,C 90.000,E1 332.871} C_DIS
LIN {X -0.059,Y -618.751,Z 1068.644,A 0.000,B 0.000,C 90.000,E1 331.847} C_DIS
LIN {X 0.191,Y -619.715,Z 1068.638,A 0.000,B 0.000,C 90.000,E1 330.795} C_DIS
LIN {X -0.083,Y -620.438,Z 1068.632,A 0.000,B 0.000,C 90.000,E1 329.793} C_DIS
LIN {X 0.189,Y -620.871,Z 1068.626,A 0.000,B 0.000,C 90.000,E1 328.742} C_DIS
LIN {X -0.072,Y -621.064,Z 1068.621,A 0.000,B 0.000,C 90.000,E1 327.740} C_DIS
LIN {X 0.320,Y -620.831,Z 1068.614,A 0.000,B 0.000,C 90.000,E1 326.421} C_DIS
LIN {X -0.117,Y -620.331,Z 1068.608,A 0.000,B 0.000,C 90.000,E1 325.435} C_DIS
LIN {X 0.135,Y -619.933,Z 1068.604,A 0.000,B 0.000,C 90.000,E1 324.642} C_DIS
LIN {X 0.137,Y -618.804,Z 1068.594,A 0.000,B 0.000,C 90.000,E1 322.844} C_DIS
LIN {X 0.113,Y -617.721,Z 1068.584,A 0.000,B 0.000,C 90.000,E1 321.045} C_DIS
LIN {X -0.338,Y -617.065,Z 1068.575,A 0.000,B 0.000,C 90.000,E1 319.542} C_DIS
LIN {X 0.100,Y -616.734,Z 1068.571,A 0.000,B 0.000,C 90.000,E1 318.728} C_DIS
LIN {X -0.228,Y -616.465,Z 1068.568,A 0.000,B 0.000,C 90.000,E1 318.243} C_DIS
LIN {X -0.096,Y -616.279,Z 1068.565,A 0.000,B 0.000,C 90.000,E1 317.715} C_DIS
LIN {X -0.075,Y -615.125,Z 1068.554,A 0.000,B 0.000,C 90.000,E1 315.648} C_DIS
LIN {X -0.022,Y -614.407,Z 1068.546,A 0.000,B 0.000,C 90.000,E1 314.352} C_DIS
LIN {X 0.291,Y -613.579,Z 1068.538,A 0.000,B 0.000,C 90.000,E1 312.771} C_DIS
LIN {X -0.115,Y -612.750,Z 1068.531,A 0.000,B 0.000,C 90.000,E1 311.515} C_DIS
LIN {X -0.089,Y -611.472,Z 1068.519,A 0.000,B 0.000,C 90.000,E1 309.439} C_DIS
LIN {X -0.181,Y -610.570,Z 1068.510,A 0.000,B 0.000,C 90.000,E1 307.890} C_DIS
LIN {X 0.106,Y -610.115,Z 1068.505,A 0.000,B 0.000,C 90.000,E1 306.824} C_DIS
LIN {X -0.386,Y -609.560,Z 1068.500,A 0.000,B 0.000,C 90.000,E1 306.091} C_DIS
LIN {X -0.115,Y -609.192,Z 1068.495,A 0.000,B 0.000,C 90.000,E1 305.025} C_DIS
LIN {X 0.152,Y -608.409,Z 1068.487,A 0.000,B 0.000,C 90.000,E1 303.706} C_DIS
LIN {X -0.213,Y -608.231,Z 1068.483,A 0.000,B 0.000,C 90.000,E1 302.959} C_DIS
LIN {X -0.113,Y -607.390,Z 1068.474,A 0.000,B 0.000,C 90.000,E1 301.386} C_DIS
LIN {X 0.164,Y -606.010,Z 1068.466,A 0.000,B 0.000,C 90.000,E1 299.795} C_DIS
LIN {X 0.232,Y -604.563,Z 1068.460,A 0.000,B 0.000,C 90.000,E1 298.743} C_DIS
LIN {X -0.007,Y -602.499,Z 1068.454,A 0.000,B 0.000,C 90.000,E1 297.719} C_DIS
LIN {X 0.075,Y -600.330,Z 1068.450,A 0.000,B 0.000,C 90.000,E1 296.924} C_DIS
LIN {X -0.143,Y -597.900,Z 1068.445,A 0.000,B 0.000,C 90.000,E1 296.155} C_DIS
LIN {X 0.236,Y -595.860,Z 1068.442,A 0.000,B 0.000,C 90.000,E1 295.591} C_DIS
LIN {X 0.015,Y -592.606,Z 1068.439,A 0.000,B 0.000,C 90.000,E1 294.951} C_DIS
LIN {X -0.131,Y -590.362,Z 1068.437,A 0.000,B 0.000,C 90.000,E1 294.567} C_DIS
LIN {X -0.049,Y -586.488,Z 1068.433,A 0.000,B 0.000,C 90.000,E1 294.027} C_DIS
LIN {X 0.254,Y -577.591,Z 1068.428,A 0.000,B 0.000,C 90.000,E1 293.078} C_DIS
LIN {X 0.053,Y -573.531,Z 1068.426,A 0.000,B 0.000,C 90.000,E1 292.717} C_DIS
LIN {X 0.182,Y -569.112,Z 1068.424,A 0.000,B 0.000,C 90.000,E1 292.333} C_DIS
LIN {X -0.199,Y -566.189,Z 1068.423,A 0.000,B 0.000,C 90.000,E1 292.153} C_DIS
LIN {X 0.076,Y -564.370,Z 1068.422,A 0.000,B 0.000,C 90.000,E1 292.025} C_DIS
LIN {X -0.066,Y -562.314,Z 1068.422,A 0.000,B 0.000,C 90.000,E1 291.950} C_DIS
LIN {X 0.102,Y -558.675,Z 1068.422,A 0.000,B 0.000,C 90.000,E1 291.844} C_DIS
LIN {X -0.345,Y -555.865,Z 1068.421,A 0.000,B 0.000,C 90.000,E1 291.844} C_DIS
LIN {X 0.202,Y -549.488,Z 1068.421,A 0.000,B 0.000,C 90.000,E1 291.770} C_DIS
LIN {X -0.027,Y -548.908,Z 1068.421,A 0.000,B 0.000,C 90.000,E1 291.770} C_DIS
LIN {X -0.150,Y -548.352,Z 1068.421,A 0.000,B 0.000,C 90.000,E1 291.716} C_DIS
LIN {X 0.171,Y -546.528,Z 1068.420,A 0.000,B 0.000,C 90.000,E1 291.535} C_DIS
LIN {X 0.264,Y -545.573,Z 1068.419,A 0.000,B 0.000,C 90.000,E1 291.408} C_DIS
LIN {X -0.071,Y -545.140,Z 1068.419,A 0.000,B 0.000,C 90.000,E1 291.354} C_DIS
LIN {X -0.231,Y -544.342,Z 1068.416,A 0.000,B 0.000,C 90.000,E1 290.918} C_DIS
LIN {X -0.128,Y -543.824,Z 1068.413,A 0.000,B 0.000,C 90.000,E1 290.301} C_DIS
LIN {X -0.295,Y -543.529,Z 1068.405,A 0.000,B 0.000,C 90.000,E1 288.906} C_DIS
LIN {X 0.101,Y -543.600,Z 1068.396,A 0.000,B 0.000,C 90.000,E1 287.166} C_DIS
LIN {X -0.253,Y -543.412,Z 1068.388,A 0.000,B 0.000,C 90.000,E1 285.788} C_DIS
LIN {X -0.096,Y -542.997,Z 1068.380,A 0.000,B 0.000,C 90.000,E1 284.356} C_DIS
LIN {X -0.092,Y -542.546,Z 1068.372,A 0.000,B 0.000,C 90.000,E1 282.939} C_DIS
LIN {X -0.139,Y -541.627,Z 1068.362,A 0.000,B 0.000,C 90.000,E1 281.243} C_DIS
LIN {X 0.232,Y -540.656,Z 1068.353,A 0.000,B 0.000,C 90.000,E1 279.500} C_DIS
LIN {X -0.021,Y -539.889,Z 1068.345,A 0.000,B 0.000,C 90.000,E1 278.106} C_DIS
LIN {X 0.230,Y -538.737,Z 1068.334,A 0.000,B 0.000,C 90.000,E1 276.087} C_DIS
LIN {X -0.132,Y -537.656,Z 1068.323,A 0.000,B 0.000,C 90.000,E1 274.131} C_DIS
LIN {X -0.032,Y -536.767,Z 1068.313,A 0.000,B 0.000,C 90.000,E1 272.407} C_DIS
LIN {X 0.015,Y -535.973,Z 1068.305,A 0.000,B 0.000,C 90.000,E1 270.974} C_DIS
LIN {X 0.037,Y -535.013,Z 1068.296,A 0.000,B 0.000,C 90.000,E1 269.255} C_DIS
LIN {X 0.049,Y -533.986,Z 1068.286,A 0.000,B 0.000,C 90.000,E1 267.535} C_DIS
LIN {X 0.042,Y -533.108,Z 1068.278,A 0.000,B 0.000,C 90.000,E1 266.102} C_DIS
LIN {X 0.079,Y -531.897,Z 1068.269,A 0.000,B 0.000,C 90.000,E1 264.375} C_DIS
LIN {X 0.124,Y -530.626,Z 1068.261,A 0.000,B 0.000,C 90.000,E1 262.932} C_DIS
LIN {X 0.111,Y -529.426,Z 1068.254,A 0.000,B 0.000,C 90.000,E1 261.781} C_DIS
LIN {X 0.204,Y -527.547,Z 1068.245,A 0.000,B 0.000,C 90.000,E1 260.038} C_DIS
LIN {X -0.184,Y -525.977,Z 1068.237,A 0.000,B 0.000,C 90.000,E1 258.634} C_DIS
LIN {X -0.083,Y -524.472,Z 1068.229,A 0.000,B 0.000,C 90.000,E1 257.173} C_DIS
LIN {X 0.107,Y -522.668,Z 1068.219,A 0.000,B 0.000,C 90.000,E1 255.408} C_DIS
LIN {X -0.116,Y -521.184,Z 1068.211,A 0.000,B 0.000,C 90.000,E1 253.976} C_DIS
LIN {X 0.273,Y -519.357,Z 1068.201,A 0.000,B 0.000,C 90.000,E1 252.181} C_DIS
LIN {X 0.010,Y -518.074,Z 1068.195,A 0.000,B 0.000,C 90.000,E1 251.040} C_DIS
LIN {X 0.114,Y -515.740,Z 1068.183,A 0.000,B 0.000,C 90.000,E1 248.975} C_DIS
LIN {X -0.199,Y -513.700,Z 1068.175,A 0.000,B 0.000,C 90.000,E1 247.539} C_DIS
LIN {X -0.184,Y -512.054,Z 1068.169,A 0.000,B 0.000,C 90.000,E1 246.357} C_DIS
LIN {X 0.123,Y -509.856,Z 1068.160,A 0.000,B 0.000,C 90.000,E1 244.845} C_DIS
LIN {X -0.075,Y -507.469,Z 1068.152,A 0.000,B 0.000,C 90.000,E1 243.384} C_DIS
LIN {X -0.016,Y -504.499,Z 1068.142,A 0.000,B 0.000,C 90.000,E1 241.591} C_DIS
LIN {X 0.092,Y -502.478,Z 1068.136,A 0.000,B 0.000,C 90.000,E1 240.383} C_DIS
LIN {X 0.223,Y -499.772,Z 1068.127,A 0.000,B 0.000,C 90.000,E1 238.869} C_DIS
LIN {X -0.274,Y -496.463,Z 1068.117,A 0.000,B 0.000,C 90.000,E1 237.120} C_DIS
LIN {X -0.155,Y -493.540,Z 1068.109,A 0.000,B 0.000,C 90.000,E1 235.595} C_DIS
LIN {X 0.060,Y -491.158,Z 1068.102,A 0.000,B 0.000,C 90.000,E1 234.356} C_DIS
LIN {X -0.037,Y -487.935,Z 1068.094,A 0.000,B 0.000,C 90.000,E1 232.844} C_DIS
LIN {X -0.064,Y -483.771,Z 1068.083,A 0.000,B 0.000,C 90.000,E1 231.009} C_DIS
LIN {X 0.195,Y -481.060,Z 1068.077,A 0.000,B 0.000,C 90.000,E1 229.747} C_DIS
LIN {X 0.069,Y -476.459,Z 1068.064,A 0.000,B 0.000,C 90.000,E1 227.595} C_DIS
LIN {X 0.046,Y -472.815,Z 1068.054,A 0.000,B 0.000,C 90.000,E1 225.729} C_DIS
LIN {X 0.084,Y -468.128,Z 1068.040,A 0.000,B 0.000,C 90.000,E1 223.218} C_DIS
LIN {X -0.197,Y -465.093,Z 1068.031,A 0.000,B 0.000,C 90.000,E1 221.676} C_DIS
LIN {X -0.182,Y -461.836,Z 1068.023,A 0.000,B 0.000,C 90.000,E1 220.092} C_DIS
LIN {X -0.137,Y -458.004,Z 1068.012,A 0.000,B 0.000,C 90.000,E1 218.177} C_DIS
LIN {X -0.190,Y -454.849,Z 1068.003,A 0.000,B 0.000,C 90.000,E1 216.583} C_DIS
LIN {X 0.136,Y -450.754,Z 1067.992,A 0.000,B 0.000,C 90.000,E1 214.612} C_DIS
LIN {X 0.243,Y -445.508,Z 1067.978,A 0.000,B 0.000,C 90.000,E1 212.005} C_DIS
LIN {X -0.056,Y -442.350,Z 1067.969,A 0.000,B 0.000,C 90.000,E1 210.413} C_DIS
LIN {X 0.143,Y -439.752,Z 1067.962,A 0.000,B 0.000,C 90.000,E1 209.077} C_DIS
LIN {X 0.181,Y -434.076,Z 1067.945,A 0.000,B 0.000,C 90.000,E1 206.104} C_DIS
LIN {X 0.220,Y -431.667,Z 1067.938,A 0.000,B 0.000,C 90.000,E1 204.771} C_DIS
LIN {X 0.190,Y -425.687,Z 1067.917,A 0.000,B 0.000,C 90.000,E1 201.099} C_DIS
LIN {X 0.164,Y -424.065,Z 1067.910,A 0.000,B 0.000,C 90.000,E1 199.758} C_DIS
LIN {X -0.055,Y -422.679,Z 1067.899,A 0.000,B 0.000,C 90.000,E1 197.764} C_DIS
LIN {X -0.095,Y -422.758,Z 1067.895,A 0.000,B 0.000,C 90.000,E1 197.094} C_DIS
LIN {X 0.146,Y -423.238,Z 1067.891,A 0.000,B 0.000,C 90.000,E1 196.386} C_DIS
LIN {X 0.103,Y -424.100,Z 1067.887,A 0.000,B 0.000,C 90.000,E1 195.717} C_DIS
LIN {X 0.012,Y -425.484,Z 1067.884,A 0.000,B 0.000,C 90.000,E1 195.064} C_DIS
LIN {X 0.089,Y -426.277,Z 1067.882,A 0.000,B 0.000,C 90.000,E1 194.717} C_DIS
LIN {X 0.047,Y -428.998,Z 1067.877,A 0.000,B 0.000,C 90.000,E1 193.883} C_DIS
LIN {X -0.070,Y -432.425,Z 1067.873,A 0.000,B 0.000,C 90.000,E1 193.063} C_DIS
LIN {X -0.039,Y -437.173,Z 1067.867,A 0.000,B 0.000,C 90.000,E1 192.063} C_DIS
LIN {X 0.101,Y -452.752,Z 1067.852,A 0.000,B 0.000,C 90.000,E1 189.265} C_DIS
LIN {X 0.147,Y -461.537,Z 1067.844,A 0.000,B 0.000,C 90.000,E1 187.814} C_DIS
LIN {X -0.071,Y -471.113,Z 1067.835,A 0.000,B 0.000,C 90.000,E1 186.258} C_DIS
LIN {X 0.056,Y -478.284,Z 1067.828,A 0.000,B 0.000,C 90.000,E1 184.992} C_DIS
LIN {X -0.188,Y -485.270,Z 1067.821,A 0.000,B 0.000,C 90.000,E1 183.784} C_DIS
LIN {X 0.124,Y -492.144,Z 1067.814,A 0.000,B 0.000,C 90.000,E1 182.522} C_DIS
LIN {X 0.235,Y -499.671,Z 1067.807,A 0.000,B 0.000,C 90.000,E1 181.146} C_DIS
LIN {X -0.044,Y -506.956,Z 1067.799,A 0.000,B 0.000,C 90.000,E1 179.828} C_DIS
LIN {X 0.229,Y -515.753,Z 1067.790,A 0.000,B 0.000,C 90.000,E1 178.167} C_DIS
LIN {X 0.046,Y -520.441,Z 1067.785,A 0.000,B 0.000,C 90.000,E1 177.306} C_DIS
LIN {X -0.127,Y -528.166,Z 1067.777,A 0.000,B 0.000,C 90.000,E1 175.869} C_DIS
LIN {X -0.157,Y -535.814,Z 1067.769,A 0.000,B 0.000,C 90.000,E1 174.432} C_DIS
LIN {X 0.279,Y -544.125,Z 1067.760,A 0.000,B 0.000,C 90.000,E1 172.818} C_DIS
LIN {X -0.235,Y -550.756,Z 1067.753,A 0.000,B 0.000,C 90.000,E1 171.602} C_DIS
LIN {X -0.109,Y -557.242,Z 1067.746,A 0.000,B 0.000,C 90.000,E1 170.330} C_DIS
LIN {X 0.072,Y -564.262,Z 1067.739,A 0.000,B 0.000,C 90.000,E1 168.926} C_DIS
LIN {X -0.093,Y -568.305,Z 1067.734,A 0.000,B 0.000,C 90.000,E1 168.117} C_DIS
LIN {X 0.020,Y -572.305,Z 1067.729,A 0.000,B 0.000,C 90.000,E1 167.285} C_DIS
LIN {X -0.089,Y -578.609,Z 1067.722,A 0.000,B 0.000,C 90.000,E1 165.936} C_DIS
LIN {X 0.043,Y -584.615,Z 1067.714,A 0.000,B 0.000,C 90.000,E1 164.574} C_DIS
LIN {X 0.021,Y -589.185,Z 1067.708,A 0.000,B 0.000,C 90.000,E1 163.504} C_DIS
LIN {X -0.197,Y -592.436,Z 1067.704,A 0.000,B 0.000,C 90.000,E1 162.725} C_DIS
LIN {X 0.062,Y -596.543,Z 1067.698,A 0.000,B 0.000,C 90.000,E1 161.638} C_DIS
LIN {X -0.084,Y -599.443,Z 1067.694,A 0.000,B 0.000,C 90.000,E1 160.859} C_DIS
LIN {X -0.089,Y -603.150,Z 1067.688,A 0.000,B 0.000,C 90.000,E1 159.806} C_DIS
LIN {X 0.254,Y -607.421,Z 1067.681,A 0.000,B 0.000,C 90.000,E1 158.465} C_DIS
LIN {X 0.140,Y -610.667,Z 1067.675,A 0.000,B 0.000,C 90.000,E1 157.433} C_DIS
LIN {X -0.304,Y -614.477,Z 1067.668,A 0.000,B 0.000,C 90.000,E1 156.177} C_DIS
LIN {X 0.137,Y -618.080,Z 1067.660,A 0.000,B 0.000,C 90.000,E1 154.845} C_DIS
LIN {X 0.102,Y -620.087,Z 1067.656,A 0.000,B 0.000,C 90.000,E1 154.076} C_DIS
LIN {X 0.101,Y -624.593,Z 1067.646,A 0.000,B 0.000,C 90.000,E1 152.281} C_DIS
LIN {X 0.153,Y -627.675,Z 1067.639,A 0.000,B 0.000,C 90.000,E1 151.001} C_DIS
LIN {X 0.004,Y -630.659,Z 1067.632,A 0.000,B 0.000,C 90.000,E1 149.744} C_DIS
LIN {X -0.252,Y -634.566,Z 1067.622,A 0.000,B 0.000,C 90.000,E1 147.995} C_DIS
LIN {X 0.045,Y -637.271,Z 1067.615,A 0.000,B 0.000,C 90.000,E1 146.707} C_DIS
LIN {X 0.246,Y -640.411,Z 1067.607,A 0.000,B 0.000,C 90.000,E1 145.182} C_DIS
LIN {X -0.016,Y -643.457,Z 1067.598,A 0.000,B 0.000,C 90.000,E1 143.703} C_DIS
LIN {X -0.191,Y -644.996,Z 1067.594,A 0.000,B 0.000,C 90.000,E1 142.970} C_DIS
LIN {X 0.106,Y -647.546,Z 1067.587,A 0.000,B 0.000,C 90.000,E1 141.698} C_DIS
LIN {X -0.275,Y -651.621,Z 1067.576,A 0.000,B 0.000,C 90.000,E1 139.747} C_DIS
LIN {X -0.112,Y -655.818,Z 1067.565,A 0.000,B 0.000,C 90.000,E1 137.757} C_DIS
LIN {X -0.349,Y -660.725,Z 1067.553,A 0.000,B 0.000,C 90.000,E1 135.567} C_DIS
LIN {X 0.028,Y -664.913,Z 1067.544,A 0.000,B 0.000,C 90.000,E1 133.824} C_DIS
LIN {X 0.016,Y -669.455,Z 1067.534,A 0.000,B 0.000,C 90.000,E1 132.123} C_DIS
LIN {X -0.192,Y -675.812,Z 1067.521,A 0.000,B 0.000,C 90.000,E1 129.725} C_DIS
LIN {X 0.142,Y -680.018,Z 1067.511,A 0.000,B 0.000,C 90.000,E1 128.016} C_DIS
LIN {X 0.093,Y -683.172,Z 1067.505,A 0.000,B 0.000,C 90.000,E1 126.824} C_DIS
LIN {X -0.046,Y -686.245,Z 1067.498,A 0.000,B 0.000,C 90.000,E1 125.644} C_DIS
LIN {X 0.437,Y -690.894,Z 1067.488,A 0.000,B 0.000,C 90.000,E1 123.706} C_DIS
LIN {X -0.173,Y -694.307,Z 1067.480,A 0.000,B 0.000,C 90.000,E1 122.339} C_DIS
LIN {X 0.212,Y -696.978,Z 1067.473,A 0.000,B 0.000,C 90.000,E1 121.131} C_DIS
LIN {X -0.316,Y -699.540,Z 1067.467,A 0.000,B 0.000,C 90.000,E1 120.001} C_DIS
LIN {X -0.128,Y -700.668,Z 1067.463,A 0.000,B 0.000,C 90.000,E1 119.283} C_DIS
LIN {X -0.199,Y -701.285,Z 1067.460,A 0.000,B 0.000,C 90.000,E1 118.821} C_DIS
LIN {X -0.230,Y -703.452,Z 1067.447,A 0.000,B 0.000,C 90.000,E1 116.488} C_DIS
LIN {X -0.013,Y -704.205,Z 1067.443,A 0.000,B 0.000,C 90.000,E1 115.771} C_DIS
LIN {X -0.109,Y -704.760,Z 1067.438,A 0.000,B 0.000,C 90.000,E1 114.847} C_DIS
LIN {X 0.178,Y -704.817,Z 1067.437,A 0.000,B 0.000,C 90.000,E1 114.591} C_DIS
LIN {X 0.108,Y -704.440,Z 1067.434,A 0.000,B 0.000,C 90.000,E1 114.131} C_DIS
LIN {X 0.106,Y -704.009,Z 1067.433,A 0.000,B 0.000,C 90.000,E1 113.898} C_DIS
LIN {X -0.255,Y -702.574,Z 1067.430,A 0.000,B 0.000,C 90.000,E1 113.462} C_DIS
LIN {X -0.116,Y -702.051,Z 1067.430,A 0.000,B 0.000,C 90.000,E1 113.334} C_DIS
LIN {X 0.156,Y -698.661,Z 1067.427,A 0.000,B 0.000,C 90.000,E1 112.845} C_DIS
LIN {X -0.354,Y -697.723,Z 1067.426,A 0.000,B 0.000,C 90.000,E1 112.770} C_DIS
LIN {X -0.225,Y -696.355,Z 1067.426,A 0.000,B 0.000,C 90.000,E1 112.642} C_DIS
LIN {X -0.095,Y -694.164,Z 1067.425,A 0.000,B 0.000,C 90.000,E1 112.514} C_DIS
LIN {X -0.140,Y -687.266,Z 1067.423,A 0.000,B 0.000,C 90.000,E1 112.206} C_DIS
LIN {X -0.369,Y -685.031,Z 1067.423,A 0.000,B 0.000,C 90.000,E1 112.153} C_DIS
LIN {X 0.013,Y -678.059,Z 1067.422,A 0.000,B 0.000,C 90.000,E1 112.025} C_DIS
LIN {X -0.264,Y -676.088,Z 1067.422,A 0.000,B 0.000,C 90.000,E1 112.025} C_DIS
LIN {X -0.292,Y -608.018,Z 1067.422,A 0.000,B 0.000,C 90.000,E1 112.025} C_DIS
LIN {X -0.103,Y -603.807,Z 1067.421,A 0.000,B 0.000,C 90.000,E1 111.844} C_DIS
LIN {X -0.012,Y -602.303,Z 1067.421,A 0.000,B 0.000,C 90.000,E1 111.770} C_DIS
LIN {X 0.306,Y -596.545,Z 1067.419,A 0.000,B 0.000,C 90.000,E1 111.408} C_DIS
LIN {X 0.207,Y -589.958,Z 1067.416,A 0.000,B 0.000,C 90.000,E1 110.918} C_DIS
LIN {X 0.297,Y -578.976,Z 1067.411,A 0.000,B 0.000,C 90.000,E1 109.993} C_DIS
LIN {X -0.086,Y -574.692,Z 1067.409,A 0.000,B 0.000,C 90.000,E1 109.685} C_DIS
LIN {X 0.166,Y -568.696,Z 1067.407,A 0.000,B 0.000,C 90.000,E1 109.214} C_DIS
LIN {X 0.128,Y -560.482,Z 1067.404,A 0.000,B 0.000,C 90.000,E1 108.725} C_DIS
LIN {X 0.090,Y -554.073,Z 1067.402,A 0.000,B 0.000,C 90.000,E1 108.362} C_DIS
LIN {X -0.231,Y -549.177,Z 1067.400,A 0.000,B 0.000,C 90.000,E1 108.055} C_DIS
LIN {X -0.210,Y -547.672,Z 1067.399,A 0.000,B 0.000,C 90.000,E1 107.873} C_DIS
LIN {X 0.269,Y -547.663,Z 1067.399,A 0.000,B 0.000,C 90.000,E1 107.819} C_DIS
LIN {X -0.290,Y -547.305,Z 1067.398,A 0.000,B 0.000,C 90.000,E1 107.583} C_DIS
LIN {X -0.285,Y -548.639,Z 1067.384,A 0.000,B 0.000,C 90.000,E1 105.190} C_DIS
LIN {X 0.283,Y -550.310,Z 1067.372,A 0.000,B 0.000,C 90.000,E1 102.883} C_DIS
LIN {X 0.112,Y -552.304,Z 1067.359,A 0.000,B 0.000,C 90.000,E1 100.658} C_DIS
LIN {X 0.228,Y -554.414,Z 1067.349,A 0.000,B 0.000,C 90.000,E1 98.690} C_DIS
LIN {X -0.272,Y -556.330,Z 1067.339,A 0.000,B 0.000,C 90.000,E1 97.068} C_DIS
LIN {X 0.236,Y -557.882,Z 1067.331,A 0.000,B 0.000,C 90.000,E1 95.625} C_DIS
LIN {X 0.078,Y -558.940,Z 1067.325,A 0.000,B 0.000,C 90.000,E1 94.531} C_DIS
LIN {X -0.023,Y -559.810,Z 1067.318,A 0.000,B 0.000,C 90.000,E1 93.154} C_DIS
LIN {X -0.082,Y -560.549,Z 1067.310,A 0.000,B 0.000,C 90.000,E1 91.776} C_DIS
LIN {X -0.170,Y -561.156,Z 1067.302,A 0.000,B 0.000,C 90.000,E1 90.401} C_DIS
LIN {X -0.146,Y -561.798,Z 1067.293,A 0.000,B 0.000,C 90.000,E1 88.740} C_DIS
LIN {X 0.125,Y -562.623,Z 1067.281,A 0.000,B 0.000,C 90.000,E1 86.502} C_DIS
LIN {X 0.128,Y -563.122,Z 1067.273,A 0.000,B 0.000,C 90.000,E1 85.122} C_DIS
LIN {X 0.138,Y -563.560,Z 1067.265,A 0.000,B 0.000,C 90.000,E1 83.742} C_DIS
LIN {X -0.105,Y -564.060,Z 1067.255,A 0.000,B 0.000,C 90.000,E1 81.837} C_DIS
LIN {X -0.166,Y -564.755,Z 1067.244,A 0.000,B 0.000,C 90.000,E1 79.916} C_DIS
LIN {X 0.135,Y -565.858,Z 1067.230,A 0.000,B 0.000,C 90.000,E1 77.409} C_DIS
LIN {X 0.187,Y -566.804,Z 1067.221,A 0.000,B 0.000,C 90.000,E1 75.755} C_DIS
LIN {X 0.158,Y -568.731,Z 1067.206,A 0.000,B 0.000,C 90.000,E1 73.015} C_DIS
LIN {X -0.130,Y -569.994,Z 1067.197,A 0.000,B 0.000,C 90.000,E1 71.402} C_DIS
